   // GBK_TO_UNICODE[37068] := 16#E9F9;
   // GBK_TO_UNICODE[37069] := 16#8F7E;
   // GBK_TO_UNICODE[37070] := 16#E9FA;
   // GBK_TO_UNICODE[37071] := 16#8F81;
   // GBK_TO_UNICODE[37072] := 16#E9FB;
   // GBK_TO_UNICODE[37073] := 16#8F82;
   // GBK_TO_UNICODE[37074] := 16#E9FC;
   // GBK_TO_UNICODE[37075] := 16#8F84;
   // GBK_TO_UNICODE[37076] := 16#E9FD;
   // GBK_TO_UNICODE[37077] := 16#8F87;
   // GBK_TO_UNICODE[37078] := 16#E9FE;
   // GBK_TO_UNICODE[37079] := 16#8F8B;
   // GBK_TO_UNICODE[37080] := 16#EA40;
   // GBK_TO_UNICODE[37081] := 16#95CC;
   // GBK_TO_UNICODE[37082] := 16#EA41;
   // GBK_TO_UNICODE[37083] := 16#95CD;
   // GBK_TO_UNICODE[37084] := 16#EA42;
   // GBK_TO_UNICODE[37085] := 16#95CE;
   // GBK_TO_UNICODE[37086] := 16#EA43;
   // GBK_TO_UNICODE[37087] := 16#95CF;
   // GBK_TO_UNICODE[37088] := 16#EA44;
   // GBK_TO_UNICODE[37089] := 16#95D0;
   // GBK_TO_UNICODE[37090] := 16#EA45;
   // GBK_TO_UNICODE[37091] := 16#95D1;
   // GBK_TO_UNICODE[37092] := 16#EA46;
   // GBK_TO_UNICODE[37093] := 16#95D2;
   // GBK_TO_UNICODE[37094] := 16#EA47;
   // GBK_TO_UNICODE[37095] := 16#95D3;
   // GBK_TO_UNICODE[37096] := 16#EA48;
   // GBK_TO_UNICODE[37097] := 16#95D4;
   // GBK_TO_UNICODE[37098] := 16#EA49;
   // GBK_TO_UNICODE[37099] := 16#95D5;
   // GBK_TO_UNICODE[37100] := 16#EA4A;
   // GBK_TO_UNICODE[37101] := 16#95D6;
   // GBK_TO_UNICODE[37102] := 16#EA4B;
   // GBK_TO_UNICODE[37103] := 16#95D7;
   // GBK_TO_UNICODE[37104] := 16#EA4C;
   // GBK_TO_UNICODE[37105] := 16#95D8;
   // GBK_TO_UNICODE[37106] := 16#EA4D;
   // GBK_TO_UNICODE[37107] := 16#95D9;
   // GBK_TO_UNICODE[37108] := 16#EA4E;
   // GBK_TO_UNICODE[37109] := 16#95DA;
   // GBK_TO_UNICODE[37110] := 16#EA4F;
   // GBK_TO_UNICODE[37111] := 16#95DB;
   // GBK_TO_UNICODE[37112] := 16#EA50;
   // GBK_TO_UNICODE[37113] := 16#95DC;
   // GBK_TO_UNICODE[37114] := 16#EA51;
   // GBK_TO_UNICODE[37115] := 16#95DD;
   // GBK_TO_UNICODE[37116] := 16#EA52;
   // GBK_TO_UNICODE[37117] := 16#95DE;
   // GBK_TO_UNICODE[37118] := 16#EA53;
   // GBK_TO_UNICODE[37119] := 16#95DF;
   // GBK_TO_UNICODE[37120] := 16#EA54;
   // GBK_TO_UNICODE[37121] := 16#95E0;
   // GBK_TO_UNICODE[37122] := 16#EA55;
   // GBK_TO_UNICODE[37123] := 16#95E1;
   // GBK_TO_UNICODE[37124] := 16#EA56;
   // GBK_TO_UNICODE[37125] := 16#95E2;
   // GBK_TO_UNICODE[37126] := 16#EA57;
   // GBK_TO_UNICODE[37127] := 16#95E3;
   // GBK_TO_UNICODE[37128] := 16#EA58;
   // GBK_TO_UNICODE[37129] := 16#95E4;
   // GBK_TO_UNICODE[37130] := 16#EA59;
   // GBK_TO_UNICODE[37131] := 16#95E5;
   // GBK_TO_UNICODE[37132] := 16#EA5A;
   // GBK_TO_UNICODE[37133] := 16#95E6;
   // GBK_TO_UNICODE[37134] := 16#EA5B;
   // GBK_TO_UNICODE[37135] := 16#95E7;
   // GBK_TO_UNICODE[37136] := 16#EA5C;
   // GBK_TO_UNICODE[37137] := 16#95EC;
   // GBK_TO_UNICODE[37138] := 16#EA5D;
   // GBK_TO_UNICODE[37139] := 16#95FF;
   // GBK_TO_UNICODE[37140] := 16#EA5E;
   // GBK_TO_UNICODE[37141] := 16#9607;
   // GBK_TO_UNICODE[37142] := 16#EA5F;
   // GBK_TO_UNICODE[37143] := 16#9613;
   // GBK_TO_UNICODE[37144] := 16#EA60;
   // GBK_TO_UNICODE[37145] := 16#9618;
   // GBK_TO_UNICODE[37146] := 16#EA61;
   // GBK_TO_UNICODE[37147] := 16#961B;
   // GBK_TO_UNICODE[37148] := 16#EA62;
   // GBK_TO_UNICODE[37149] := 16#961E;
   // GBK_TO_UNICODE[37150] := 16#EA63;
   // GBK_TO_UNICODE[37151] := 16#9620;
   // GBK_TO_UNICODE[37152] := 16#EA64;
   // GBK_TO_UNICODE[37153] := 16#9623;
   // GBK_TO_UNICODE[37154] := 16#EA65;
   // GBK_TO_UNICODE[37155] := 16#9624;
   // GBK_TO_UNICODE[37156] := 16#EA66;
   // GBK_TO_UNICODE[37157] := 16#9625;
   // GBK_TO_UNICODE[37158] := 16#EA67;
   // GBK_TO_UNICODE[37159] := 16#9626;
   // GBK_TO_UNICODE[37160] := 16#EA68;
   // GBK_TO_UNICODE[37161] := 16#9627;
   // GBK_TO_UNICODE[37162] := 16#EA69;
   // GBK_TO_UNICODE[37163] := 16#9628;
   // GBK_TO_UNICODE[37164] := 16#EA6A;
   // GBK_TO_UNICODE[37165] := 16#9629;
   // GBK_TO_UNICODE[37166] := 16#EA6B;
   // GBK_TO_UNICODE[37167] := 16#962B;
   // GBK_TO_UNICODE[37168] := 16#EA6C;
   // GBK_TO_UNICODE[37169] := 16#962C;
   // GBK_TO_UNICODE[37170] := 16#EA6D;
   // GBK_TO_UNICODE[37171] := 16#962D;
   // GBK_TO_UNICODE[37172] := 16#EA6E;
   // GBK_TO_UNICODE[37173] := 16#962F;
   // GBK_TO_UNICODE[37174] := 16#EA6F;
   // GBK_TO_UNICODE[37175] := 16#9630;
   // GBK_TO_UNICODE[37176] := 16#EA70;
   // GBK_TO_UNICODE[37177] := 16#9637;
   // GBK_TO_UNICODE[37178] := 16#EA71;
   // GBK_TO_UNICODE[37179] := 16#9638;
   // GBK_TO_UNICODE[37180] := 16#EA72;
   // GBK_TO_UNICODE[37181] := 16#9639;
   // GBK_TO_UNICODE[37182] := 16#EA73;
   // GBK_TO_UNICODE[37183] := 16#963A;
   // GBK_TO_UNICODE[37184] := 16#EA74;
   // GBK_TO_UNICODE[37185] := 16#963E;
   // GBK_TO_UNICODE[37186] := 16#EA75;
   // GBK_TO_UNICODE[37187] := 16#9641;
   // GBK_TO_UNICODE[37188] := 16#EA76;
   // GBK_TO_UNICODE[37189] := 16#9643;
   // GBK_TO_UNICODE[37190] := 16#EA77;
   // GBK_TO_UNICODE[37191] := 16#964A;
   // GBK_TO_UNICODE[37192] := 16#EA78;
   // GBK_TO_UNICODE[37193] := 16#964E;
   // GBK_TO_UNICODE[37194] := 16#EA79;
   // GBK_TO_UNICODE[37195] := 16#964F;
   // GBK_TO_UNICODE[37196] := 16#EA7A;
   // GBK_TO_UNICODE[37197] := 16#9651;
   // GBK_TO_UNICODE[37198] := 16#EA7B;
   // GBK_TO_UNICODE[37199] := 16#9652;
   // GBK_TO_UNICODE[37200] := 16#EA7C;
   // GBK_TO_UNICODE[37201] := 16#9653;
   // GBK_TO_UNICODE[37202] := 16#EA7D;
   // GBK_TO_UNICODE[37203] := 16#9656;
   // GBK_TO_UNICODE[37204] := 16#EA7E;
   // GBK_TO_UNICODE[37205] := 16#9657;
   // GBK_TO_UNICODE[37206] := 16#EA80;
   // GBK_TO_UNICODE[37207] := 16#9658;
   // GBK_TO_UNICODE[37208] := 16#EA81;
   // GBK_TO_UNICODE[37209] := 16#9659;
   // GBK_TO_UNICODE[37210] := 16#EA82;
   // GBK_TO_UNICODE[37211] := 16#965A;
   // GBK_TO_UNICODE[37212] := 16#EA83;
   // GBK_TO_UNICODE[37213] := 16#965C;
   // GBK_TO_UNICODE[37214] := 16#EA84;
   // GBK_TO_UNICODE[37215] := 16#965D;
   // GBK_TO_UNICODE[37216] := 16#EA85;
   // GBK_TO_UNICODE[37217] := 16#965E;
   // GBK_TO_UNICODE[37218] := 16#EA86;
   // GBK_TO_UNICODE[37219] := 16#9660;
   // GBK_TO_UNICODE[37220] := 16#EA87;
   // GBK_TO_UNICODE[37221] := 16#9663;
   // GBK_TO_UNICODE[37222] := 16#EA88;
   // GBK_TO_UNICODE[37223] := 16#9665;
   // GBK_TO_UNICODE[37224] := 16#EA89;
   // GBK_TO_UNICODE[37225] := 16#9666;
   // GBK_TO_UNICODE[37226] := 16#EA8A;
   // GBK_TO_UNICODE[37227] := 16#966B;
   // GBK_TO_UNICODE[37228] := 16#EA8B;
   // GBK_TO_UNICODE[37229] := 16#966D;
   // GBK_TO_UNICODE[37230] := 16#EA8C;
   // GBK_TO_UNICODE[37231] := 16#966E;
   // GBK_TO_UNICODE[37232] := 16#EA8D;
   // GBK_TO_UNICODE[37233] := 16#966F;
   // GBK_TO_UNICODE[37234] := 16#EA8E;
   // GBK_TO_UNICODE[37235] := 16#9670;
   // GBK_TO_UNICODE[37236] := 16#EA8F;
   // GBK_TO_UNICODE[37237] := 16#9671;
   // GBK_TO_UNICODE[37238] := 16#EA90;
   // GBK_TO_UNICODE[37239] := 16#9673;
   // GBK_TO_UNICODE[37240] := 16#EA91;
   // GBK_TO_UNICODE[37241] := 16#9678;
   // GBK_TO_UNICODE[37242] := 16#EA92;
   // GBK_TO_UNICODE[37243] := 16#9679;
   // GBK_TO_UNICODE[37244] := 16#EA93;
   // GBK_TO_UNICODE[37245] := 16#967A;
   // GBK_TO_UNICODE[37246] := 16#EA94;
   // GBK_TO_UNICODE[37247] := 16#967B;
   // GBK_TO_UNICODE[37248] := 16#EA95;
   // GBK_TO_UNICODE[37249] := 16#967C;
   // GBK_TO_UNICODE[37250] := 16#EA96;
   // GBK_TO_UNICODE[37251] := 16#967D;
   // GBK_TO_UNICODE[37252] := 16#EA97;
   // GBK_TO_UNICODE[37253] := 16#967E;
   // GBK_TO_UNICODE[37254] := 16#EA98;
   // GBK_TO_UNICODE[37255] := 16#967F;
   // GBK_TO_UNICODE[37256] := 16#EA99;
   // GBK_TO_UNICODE[37257] := 16#9680;
   // GBK_TO_UNICODE[37258] := 16#EA9A;
   // GBK_TO_UNICODE[37259] := 16#9681;
   // GBK_TO_UNICODE[37260] := 16#EA9B;
   // GBK_TO_UNICODE[37261] := 16#9682;
   // GBK_TO_UNICODE[37262] := 16#EA9C;
   // GBK_TO_UNICODE[37263] := 16#9683;
   // GBK_TO_UNICODE[37264] := 16#EA9D;
   // GBK_TO_UNICODE[37265] := 16#9684;
   // GBK_TO_UNICODE[37266] := 16#EA9E;
   // GBK_TO_UNICODE[37267] := 16#9687;
   // GBK_TO_UNICODE[37268] := 16#EA9F;
   // GBK_TO_UNICODE[37269] := 16#9689;
   // GBK_TO_UNICODE[37270] := 16#EAA0;
   // GBK_TO_UNICODE[37271] := 16#968A;
   // GBK_TO_UNICODE[37272] := 16#EAA1;
   // GBK_TO_UNICODE[37273] := 16#8F8D;
   // GBK_TO_UNICODE[37274] := 16#EAA2;
   // GBK_TO_UNICODE[37275] := 16#8F8E;
   // GBK_TO_UNICODE[37276] := 16#EAA3;
   // GBK_TO_UNICODE[37277] := 16#8F8F;
   // GBK_TO_UNICODE[37278] := 16#EAA4;
   // GBK_TO_UNICODE[37279] := 16#8F98;
   // GBK_TO_UNICODE[37280] := 16#EAA5;
   // GBK_TO_UNICODE[37281] := 16#8F9A;
   // GBK_TO_UNICODE[37282] := 16#EAA6;
   // GBK_TO_UNICODE[37283] := 16#8ECE;
   // GBK_TO_UNICODE[37284] := 16#EAA7;
   // GBK_TO_UNICODE[37285] := 16#620B;
   // GBK_TO_UNICODE[37286] := 16#EAA8;
   // GBK_TO_UNICODE[37287] := 16#6217;
   // GBK_TO_UNICODE[37288] := 16#EAA9;
   // GBK_TO_UNICODE[37289] := 16#621B;
   // GBK_TO_UNICODE[37290] := 16#EAAA;
   // GBK_TO_UNICODE[37291] := 16#621F;
   // GBK_TO_UNICODE[37292] := 16#EAAB;
   // GBK_TO_UNICODE[37293] := 16#6222;
   // GBK_TO_UNICODE[37294] := 16#EAAC;
   // GBK_TO_UNICODE[37295] := 16#6221;
   // GBK_TO_UNICODE[37296] := 16#EAAD;
   // GBK_TO_UNICODE[37297] := 16#6225;
   // GBK_TO_UNICODE[37298] := 16#EAAE;
   // GBK_TO_UNICODE[37299] := 16#6224;
   // GBK_TO_UNICODE[37300] := 16#EAAF;
   // GBK_TO_UNICODE[37301] := 16#622C;
   // GBK_TO_UNICODE[37302] := 16#EAB0;
   // GBK_TO_UNICODE[37303] := 16#81E7;
   // GBK_TO_UNICODE[37304] := 16#EAB1;
   // GBK_TO_UNICODE[37305] := 16#74EF;
   // GBK_TO_UNICODE[37306] := 16#EAB2;
   // GBK_TO_UNICODE[37307] := 16#74F4;
   // GBK_TO_UNICODE[37308] := 16#EAB3;
   // GBK_TO_UNICODE[37309] := 16#74FF;
   // GBK_TO_UNICODE[37310] := 16#EAB4;
   // GBK_TO_UNICODE[37311] := 16#750F;
   // GBK_TO_UNICODE[37312] := 16#EAB5;
   // GBK_TO_UNICODE[37313] := 16#7511;
   // GBK_TO_UNICODE[37314] := 16#EAB6;
   // GBK_TO_UNICODE[37315] := 16#7513;
   // GBK_TO_UNICODE[37316] := 16#EAB7;
   // GBK_TO_UNICODE[37317] := 16#6534;
   // GBK_TO_UNICODE[37318] := 16#EAB8;
   // GBK_TO_UNICODE[37319] := 16#65EE;
   // GBK_TO_UNICODE[37320] := 16#EAB9;
   // GBK_TO_UNICODE[37321] := 16#65EF;
   // GBK_TO_UNICODE[37322] := 16#EABA;
   // GBK_TO_UNICODE[37323] := 16#65F0;
   // GBK_TO_UNICODE[37324] := 16#EABB;
   // GBK_TO_UNICODE[37325] := 16#660A;
   // GBK_TO_UNICODE[37326] := 16#EABC;
   // GBK_TO_UNICODE[37327] := 16#6619;
   // GBK_TO_UNICODE[37328] := 16#EABD;
   // GBK_TO_UNICODE[37329] := 16#6772;
   // GBK_TO_UNICODE[37330] := 16#EABE;
   // GBK_TO_UNICODE[37331] := 16#6603;
   // GBK_TO_UNICODE[37332] := 16#EABF;
   // GBK_TO_UNICODE[37333] := 16#6615;
   // GBK_TO_UNICODE[37334] := 16#EAC0;
   // GBK_TO_UNICODE[37335] := 16#6600;
   // GBK_TO_UNICODE[37336] := 16#EAC1;
   // GBK_TO_UNICODE[37337] := 16#7085;
   // GBK_TO_UNICODE[37338] := 16#EAC2;
   // GBK_TO_UNICODE[37339] := 16#66F7;
   // GBK_TO_UNICODE[37340] := 16#EAC3;
   // GBK_TO_UNICODE[37341] := 16#661D;
   // GBK_TO_UNICODE[37342] := 16#EAC4;
   // GBK_TO_UNICODE[37343] := 16#6634;
   // GBK_TO_UNICODE[37344] := 16#EAC5;
   // GBK_TO_UNICODE[37345] := 16#6631;
   // GBK_TO_UNICODE[37346] := 16#EAC6;
   // GBK_TO_UNICODE[37347] := 16#6636;
   // GBK_TO_UNICODE[37348] := 16#EAC7;
   // GBK_TO_UNICODE[37349] := 16#6635;
   // GBK_TO_UNICODE[37350] := 16#EAC8;
   // GBK_TO_UNICODE[37351] := 16#8006;
   // GBK_TO_UNICODE[37352] := 16#EAC9;
   // GBK_TO_UNICODE[37353] := 16#665F;
   // GBK_TO_UNICODE[37354] := 16#EACA;
   // GBK_TO_UNICODE[37355] := 16#6654;
   // GBK_TO_UNICODE[37356] := 16#EACB;
   // GBK_TO_UNICODE[37357] := 16#6641;
   // GBK_TO_UNICODE[37358] := 16#EACC;
   // GBK_TO_UNICODE[37359] := 16#664F;
   // GBK_TO_UNICODE[37360] := 16#EACD;
   // GBK_TO_UNICODE[37361] := 16#6656;
   // GBK_TO_UNICODE[37362] := 16#EACE;
   // GBK_TO_UNICODE[37363] := 16#6661;
   // GBK_TO_UNICODE[37364] := 16#EACF;
   // GBK_TO_UNICODE[37365] := 16#6657;
   // GBK_TO_UNICODE[37366] := 16#EAD0;
   // GBK_TO_UNICODE[37367] := 16#6677;
   // GBK_TO_UNICODE[37368] := 16#EAD1;
   // GBK_TO_UNICODE[37369] := 16#6684;
   // GBK_TO_UNICODE[37370] := 16#EAD2;
   // GBK_TO_UNICODE[37371] := 16#668C;
   // GBK_TO_UNICODE[37372] := 16#EAD3;
   // GBK_TO_UNICODE[37373] := 16#66A7;
   // GBK_TO_UNICODE[37374] := 16#EAD4;
   // GBK_TO_UNICODE[37375] := 16#669D;
   // GBK_TO_UNICODE[37376] := 16#EAD5;
   // GBK_TO_UNICODE[37377] := 16#66BE;
   // GBK_TO_UNICODE[37378] := 16#EAD6;
   // GBK_TO_UNICODE[37379] := 16#66DB;
   // GBK_TO_UNICODE[37380] := 16#EAD7;
   // GBK_TO_UNICODE[37381] := 16#66DC;
   // GBK_TO_UNICODE[37382] := 16#EAD8;
   // GBK_TO_UNICODE[37383] := 16#66E6;
   // GBK_TO_UNICODE[37384] := 16#EAD9;
   // GBK_TO_UNICODE[37385] := 16#66E9;
   // GBK_TO_UNICODE[37386] := 16#EADA;
   // GBK_TO_UNICODE[37387] := 16#8D32;
   // GBK_TO_UNICODE[37388] := 16#EADB;
   // GBK_TO_UNICODE[37389] := 16#8D33;
   // GBK_TO_UNICODE[37390] := 16#EADC;
   // GBK_TO_UNICODE[37391] := 16#8D36;
   // GBK_TO_UNICODE[37392] := 16#EADD;
   // GBK_TO_UNICODE[37393] := 16#8D3B;
   // GBK_TO_UNICODE[37394] := 16#EADE;
   // GBK_TO_UNICODE[37395] := 16#8D3D;
   // GBK_TO_UNICODE[37396] := 16#EADF;
   // GBK_TO_UNICODE[37397] := 16#8D40;
   // GBK_TO_UNICODE[37398] := 16#EAE0;
   // GBK_TO_UNICODE[37399] := 16#8D45;
   // GBK_TO_UNICODE[37400] := 16#EAE1;
   // GBK_TO_UNICODE[37401] := 16#8D46;
   // GBK_TO_UNICODE[37402] := 16#EAE2;
   // GBK_TO_UNICODE[37403] := 16#8D48;
   // GBK_TO_UNICODE[37404] := 16#EAE3;
   // GBK_TO_UNICODE[37405] := 16#8D49;
   // GBK_TO_UNICODE[37406] := 16#EAE4;
   // GBK_TO_UNICODE[37407] := 16#8D47;
   // GBK_TO_UNICODE[37408] := 16#EAE5;
   // GBK_TO_UNICODE[37409] := 16#8D4D;
   // GBK_TO_UNICODE[37410] := 16#EAE6;
   // GBK_TO_UNICODE[37411] := 16#8D55;
   // GBK_TO_UNICODE[37412] := 16#EAE7;
   // GBK_TO_UNICODE[37413] := 16#8D59;
   // GBK_TO_UNICODE[37414] := 16#EAE8;
   // GBK_TO_UNICODE[37415] := 16#89C7;
   // GBK_TO_UNICODE[37416] := 16#EAE9;
   // GBK_TO_UNICODE[37417] := 16#89CA;
   // GBK_TO_UNICODE[37418] := 16#EAEA;
   // GBK_TO_UNICODE[37419] := 16#89CB;
   // GBK_TO_UNICODE[37420] := 16#EAEB;
   // GBK_TO_UNICODE[37421] := 16#89CC;
   // GBK_TO_UNICODE[37422] := 16#EAEC;
   // GBK_TO_UNICODE[37423] := 16#89CE;
   // GBK_TO_UNICODE[37424] := 16#EAED;
   // GBK_TO_UNICODE[37425] := 16#89CF;
   // GBK_TO_UNICODE[37426] := 16#EAEE;
   // GBK_TO_UNICODE[37427] := 16#89D0;
   // GBK_TO_UNICODE[37428] := 16#EAEF;
   // GBK_TO_UNICODE[37429] := 16#89D1;
   // GBK_TO_UNICODE[37430] := 16#EAF0;
   // GBK_TO_UNICODE[37431] := 16#726E;
   // GBK_TO_UNICODE[37432] := 16#EAF1;
   // GBK_TO_UNICODE[37433] := 16#729F;
   // GBK_TO_UNICODE[37434] := 16#EAF2;
   // GBK_TO_UNICODE[37435] := 16#725D;
   // GBK_TO_UNICODE[37436] := 16#EAF3;
   // GBK_TO_UNICODE[37437] := 16#7266;
   // GBK_TO_UNICODE[37438] := 16#EAF4;
   // GBK_TO_UNICODE[37439] := 16#726F;
   // GBK_TO_UNICODE[37440] := 16#EAF5;
   // GBK_TO_UNICODE[37441] := 16#727E;
   // GBK_TO_UNICODE[37442] := 16#EAF6;
   // GBK_TO_UNICODE[37443] := 16#727F;
   // GBK_TO_UNICODE[37444] := 16#EAF7;
   // GBK_TO_UNICODE[37445] := 16#7284;
   // GBK_TO_UNICODE[37446] := 16#EAF8;
   // GBK_TO_UNICODE[37447] := 16#728B;
   // GBK_TO_UNICODE[37448] := 16#EAF9;
   // GBK_TO_UNICODE[37449] := 16#728D;
   // GBK_TO_UNICODE[37450] := 16#EAFA;
   // GBK_TO_UNICODE[37451] := 16#728F;
   // GBK_TO_UNICODE[37452] := 16#EAFB;
   // GBK_TO_UNICODE[37453] := 16#7292;
   // GBK_TO_UNICODE[37454] := 16#EAFC;
   // GBK_TO_UNICODE[37455] := 16#6308;
   // GBK_TO_UNICODE[37456] := 16#EAFD;
   // GBK_TO_UNICODE[37457] := 16#6332;
   // GBK_TO_UNICODE[37458] := 16#EAFE;
   // GBK_TO_UNICODE[37459] := 16#63B0;
   // GBK_TO_UNICODE[37460] := 16#EB40;
   // GBK_TO_UNICODE[37461] := 16#968C;
   // GBK_TO_UNICODE[37462] := 16#EB41;
   // GBK_TO_UNICODE[37463] := 16#968E;
   // GBK_TO_UNICODE[37464] := 16#EB42;
   // GBK_TO_UNICODE[37465] := 16#9691;
   // GBK_TO_UNICODE[37466] := 16#EB43;
   // GBK_TO_UNICODE[37467] := 16#9692;
   // GBK_TO_UNICODE[37468] := 16#EB44;
   // GBK_TO_UNICODE[37469] := 16#9693;
   // GBK_TO_UNICODE[37470] := 16#EB45;
   // GBK_TO_UNICODE[37471] := 16#9695;
   // GBK_TO_UNICODE[37472] := 16#EB46;
   // GBK_TO_UNICODE[37473] := 16#9696;
   // GBK_TO_UNICODE[37474] := 16#EB47;
   // GBK_TO_UNICODE[37475] := 16#969A;
   // GBK_TO_UNICODE[37476] := 16#EB48;
   // GBK_TO_UNICODE[37477] := 16#969B;
   // GBK_TO_UNICODE[37478] := 16#EB49;
   // GBK_TO_UNICODE[37479] := 16#969D;
   // GBK_TO_UNICODE[37480] := 16#EB4A;
   // GBK_TO_UNICODE[37481] := 16#969E;
   // GBK_TO_UNICODE[37482] := 16#EB4B;
   // GBK_TO_UNICODE[37483] := 16#969F;
   // GBK_TO_UNICODE[37484] := 16#EB4C;
   // GBK_TO_UNICODE[37485] := 16#96A0;
   // GBK_TO_UNICODE[37486] := 16#EB4D;
   // GBK_TO_UNICODE[37487] := 16#96A1;
   // GBK_TO_UNICODE[37488] := 16#EB4E;
   // GBK_TO_UNICODE[37489] := 16#96A2;
   // GBK_TO_UNICODE[37490] := 16#EB4F;
   // GBK_TO_UNICODE[37491] := 16#96A3;
   // GBK_TO_UNICODE[37492] := 16#EB50;
   // GBK_TO_UNICODE[37493] := 16#96A4;
   // GBK_TO_UNICODE[37494] := 16#EB51;
   // GBK_TO_UNICODE[37495] := 16#96A5;
   // GBK_TO_UNICODE[37496] := 16#EB52;
   // GBK_TO_UNICODE[37497] := 16#96A6;
   // GBK_TO_UNICODE[37498] := 16#EB53;
   // GBK_TO_UNICODE[37499] := 16#96A8;
   // GBK_TO_UNICODE[37500] := 16#EB54;
   // GBK_TO_UNICODE[37501] := 16#96A9;
   // GBK_TO_UNICODE[37502] := 16#EB55;
   // GBK_TO_UNICODE[37503] := 16#96AA;
   // GBK_TO_UNICODE[37504] := 16#EB56;
   // GBK_TO_UNICODE[37505] := 16#96AB;
   // GBK_TO_UNICODE[37506] := 16#EB57;
   // GBK_TO_UNICODE[37507] := 16#96AC;
   // GBK_TO_UNICODE[37508] := 16#EB58;
   // GBK_TO_UNICODE[37509] := 16#96AD;
   // GBK_TO_UNICODE[37510] := 16#EB59;
   // GBK_TO_UNICODE[37511] := 16#96AE;
   // GBK_TO_UNICODE[37512] := 16#EB5A;
   // GBK_TO_UNICODE[37513] := 16#96AF;
   // GBK_TO_UNICODE[37514] := 16#EB5B;
   // GBK_TO_UNICODE[37515] := 16#96B1;
   // GBK_TO_UNICODE[37516] := 16#EB5C;
   // GBK_TO_UNICODE[37517] := 16#96B2;
   // GBK_TO_UNICODE[37518] := 16#EB5D;
   // GBK_TO_UNICODE[37519] := 16#96B4;
   // GBK_TO_UNICODE[37520] := 16#EB5E;
   // GBK_TO_UNICODE[37521] := 16#96B5;
   // GBK_TO_UNICODE[37522] := 16#EB5F;
   // GBK_TO_UNICODE[37523] := 16#96B7;
   // GBK_TO_UNICODE[37524] := 16#EB60;
   // GBK_TO_UNICODE[37525] := 16#96B8;
   // GBK_TO_UNICODE[37526] := 16#EB61;
   // GBK_TO_UNICODE[37527] := 16#96BA;
   // GBK_TO_UNICODE[37528] := 16#EB62;
   // GBK_TO_UNICODE[37529] := 16#96BB;
   // GBK_TO_UNICODE[37530] := 16#EB63;
   // GBK_TO_UNICODE[37531] := 16#96BF;
   // GBK_TO_UNICODE[37532] := 16#EB64;
   // GBK_TO_UNICODE[37533] := 16#96C2;
   // GBK_TO_UNICODE[37534] := 16#EB65;
   // GBK_TO_UNICODE[37535] := 16#96C3;
   // GBK_TO_UNICODE[37536] := 16#EB66;
   // GBK_TO_UNICODE[37537] := 16#96C8;
   // GBK_TO_UNICODE[37538] := 16#EB67;
   // GBK_TO_UNICODE[37539] := 16#96CA;
   // GBK_TO_UNICODE[37540] := 16#EB68;
   // GBK_TO_UNICODE[37541] := 16#96CB;
   // GBK_TO_UNICODE[37542] := 16#EB69;
   // GBK_TO_UNICODE[37543] := 16#96D0;
   // GBK_TO_UNICODE[37544] := 16#EB6A;
   // GBK_TO_UNICODE[37545] := 16#96D1;
   // GBK_TO_UNICODE[37546] := 16#EB6B;
   // GBK_TO_UNICODE[37547] := 16#96D3;
   // GBK_TO_UNICODE[37548] := 16#EB6C;
   // GBK_TO_UNICODE[37549] := 16#96D4;
   // GBK_TO_UNICODE[37550] := 16#EB6D;
   // GBK_TO_UNICODE[37551] := 16#96D6;
   // GBK_TO_UNICODE[37552] := 16#EB6E;
   // GBK_TO_UNICODE[37553] := 16#96D7;
   // GBK_TO_UNICODE[37554] := 16#EB6F;
   // GBK_TO_UNICODE[37555] := 16#96D8;
   // GBK_TO_UNICODE[37556] := 16#EB70;
   // GBK_TO_UNICODE[37557] := 16#96D9;
   // GBK_TO_UNICODE[37558] := 16#EB71;
   // GBK_TO_UNICODE[37559] := 16#96DA;
   // GBK_TO_UNICODE[37560] := 16#EB72;
   // GBK_TO_UNICODE[37561] := 16#96DB;
   // GBK_TO_UNICODE[37562] := 16#EB73;
   // GBK_TO_UNICODE[37563] := 16#96DC;
   // GBK_TO_UNICODE[37564] := 16#EB74;
   // GBK_TO_UNICODE[37565] := 16#96DD;
   // GBK_TO_UNICODE[37566] := 16#EB75;
   // GBK_TO_UNICODE[37567] := 16#96DE;
   // GBK_TO_UNICODE[37568] := 16#EB76;
   // GBK_TO_UNICODE[37569] := 16#96DF;
   // GBK_TO_UNICODE[37570] := 16#EB77;
   // GBK_TO_UNICODE[37571] := 16#96E1;
   // GBK_TO_UNICODE[37572] := 16#EB78;
   // GBK_TO_UNICODE[37573] := 16#96E2;
   // GBK_TO_UNICODE[37574] := 16#EB79;
   // GBK_TO_UNICODE[37575] := 16#96E3;
   // GBK_TO_UNICODE[37576] := 16#EB7A;
   // GBK_TO_UNICODE[37577] := 16#96E4;
   // GBK_TO_UNICODE[37578] := 16#EB7B;
   // GBK_TO_UNICODE[37579] := 16#96E5;
   // GBK_TO_UNICODE[37580] := 16#EB7C;
   // GBK_TO_UNICODE[37581] := 16#96E6;
   // GBK_TO_UNICODE[37582] := 16#EB7D;
   // GBK_TO_UNICODE[37583] := 16#96E7;
   // GBK_TO_UNICODE[37584] := 16#EB7E;
   // GBK_TO_UNICODE[37585] := 16#96EB;
   // GBK_TO_UNICODE[37586] := 16#EB80;
   // GBK_TO_UNICODE[37587] := 16#96EC;
   // GBK_TO_UNICODE[37588] := 16#EB81;
   // GBK_TO_UNICODE[37589] := 16#96ED;
   // GBK_TO_UNICODE[37590] := 16#EB82;
   // GBK_TO_UNICODE[37591] := 16#96EE;
   // GBK_TO_UNICODE[37592] := 16#EB83;
   // GBK_TO_UNICODE[37593] := 16#96F0;
   // GBK_TO_UNICODE[37594] := 16#EB84;
   // GBK_TO_UNICODE[37595] := 16#96F1;
   // GBK_TO_UNICODE[37596] := 16#EB85;
   // GBK_TO_UNICODE[37597] := 16#96F2;
   // GBK_TO_UNICODE[37598] := 16#EB86;
   // GBK_TO_UNICODE[37599] := 16#96F4;
   // GBK_TO_UNICODE[37600] := 16#EB87;
   // GBK_TO_UNICODE[37601] := 16#96F5;
   // GBK_TO_UNICODE[37602] := 16#EB88;
   // GBK_TO_UNICODE[37603] := 16#96F8;
   // GBK_TO_UNICODE[37604] := 16#EB89;
   // GBK_TO_UNICODE[37605] := 16#96FA;
   // GBK_TO_UNICODE[37606] := 16#EB8A;
   // GBK_TO_UNICODE[37607] := 16#96FB;
   // GBK_TO_UNICODE[37608] := 16#EB8B;
   // GBK_TO_UNICODE[37609] := 16#96FC;
   // GBK_TO_UNICODE[37610] := 16#EB8C;
   // GBK_TO_UNICODE[37611] := 16#96FD;
   // GBK_TO_UNICODE[37612] := 16#EB8D;
   // GBK_TO_UNICODE[37613] := 16#96FF;
   // GBK_TO_UNICODE[37614] := 16#EB8E;
   // GBK_TO_UNICODE[37615] := 16#9702;
   // GBK_TO_UNICODE[37616] := 16#EB8F;
   // GBK_TO_UNICODE[37617] := 16#9703;
   // GBK_TO_UNICODE[37618] := 16#EB90;
   // GBK_TO_UNICODE[37619] := 16#9705;
   // GBK_TO_UNICODE[37620] := 16#EB91;
   // GBK_TO_UNICODE[37621] := 16#970A;
   // GBK_TO_UNICODE[37622] := 16#EB92;
   // GBK_TO_UNICODE[37623] := 16#970B;
   // GBK_TO_UNICODE[37624] := 16#EB93;
   // GBK_TO_UNICODE[37625] := 16#970C;
   // GBK_TO_UNICODE[37626] := 16#EB94;
   // GBK_TO_UNICODE[37627] := 16#9710;
   // GBK_TO_UNICODE[37628] := 16#EB95;
   // GBK_TO_UNICODE[37629] := 16#9711;
   // GBK_TO_UNICODE[37630] := 16#EB96;
   // GBK_TO_UNICODE[37631] := 16#9712;
   // GBK_TO_UNICODE[37632] := 16#EB97;
   // GBK_TO_UNICODE[37633] := 16#9714;
   // GBK_TO_UNICODE[37634] := 16#EB98;
   // GBK_TO_UNICODE[37635] := 16#9715;
   // GBK_TO_UNICODE[37636] := 16#EB99;
   // GBK_TO_UNICODE[37637] := 16#9717;
   // GBK_TO_UNICODE[37638] := 16#EB9A;
   // GBK_TO_UNICODE[37639] := 16#9718;
   // GBK_TO_UNICODE[37640] := 16#EB9B;
   // GBK_TO_UNICODE[37641] := 16#9719;
   // GBK_TO_UNICODE[37642] := 16#EB9C;
   // GBK_TO_UNICODE[37643] := 16#971A;
   // GBK_TO_UNICODE[37644] := 16#EB9D;
   // GBK_TO_UNICODE[37645] := 16#971B;
   // GBK_TO_UNICODE[37646] := 16#EB9E;
   // GBK_TO_UNICODE[37647] := 16#971D;
   // GBK_TO_UNICODE[37648] := 16#EB9F;
   // GBK_TO_UNICODE[37649] := 16#971F;
   // GBK_TO_UNICODE[37650] := 16#EBA0;
   // GBK_TO_UNICODE[37651] := 16#9720;
   // GBK_TO_UNICODE[37652] := 16#EBA1;
   // GBK_TO_UNICODE[37653] := 16#643F;
   // GBK_TO_UNICODE[37654] := 16#EBA2;
   // GBK_TO_UNICODE[37655] := 16#64D8;
   // GBK_TO_UNICODE[37656] := 16#EBA3;
   // GBK_TO_UNICODE[37657] := 16#8004;
   // GBK_TO_UNICODE[37658] := 16#EBA4;
   // GBK_TO_UNICODE[37659] := 16#6BEA;
   // GBK_TO_UNICODE[37660] := 16#EBA5;
   // GBK_TO_UNICODE[37661] := 16#6BF3;
   // GBK_TO_UNICODE[37662] := 16#EBA6;
   // GBK_TO_UNICODE[37663] := 16#6BFD;
   // GBK_TO_UNICODE[37664] := 16#EBA7;
   // GBK_TO_UNICODE[37665] := 16#6BF5;
   // GBK_TO_UNICODE[37666] := 16#EBA8;
   // GBK_TO_UNICODE[37667] := 16#6BF9;
   // GBK_TO_UNICODE[37668] := 16#EBA9;
   // GBK_TO_UNICODE[37669] := 16#6C05;
   // GBK_TO_UNICODE[37670] := 16#EBAA;
   // GBK_TO_UNICODE[37671] := 16#6C07;
   // GBK_TO_UNICODE[37672] := 16#EBAB;
   // GBK_TO_UNICODE[37673] := 16#6C06;
   // GBK_TO_UNICODE[37674] := 16#EBAC;
   // GBK_TO_UNICODE[37675] := 16#6C0D;
   // GBK_TO_UNICODE[37676] := 16#EBAD;
   // GBK_TO_UNICODE[37677] := 16#6C15;
   // GBK_TO_UNICODE[37678] := 16#EBAE;
   // GBK_TO_UNICODE[37679] := 16#6C18;
   // GBK_TO_UNICODE[37680] := 16#EBAF;
   // GBK_TO_UNICODE[37681] := 16#6C19;
   // GBK_TO_UNICODE[37682] := 16#EBB0;
   // GBK_TO_UNICODE[37683] := 16#6C1A;
   // GBK_TO_UNICODE[37684] := 16#EBB1;
   // GBK_TO_UNICODE[37685] := 16#6C21;
   // GBK_TO_UNICODE[37686] := 16#EBB2;
   // GBK_TO_UNICODE[37687] := 16#6C29;
   // GBK_TO_UNICODE[37688] := 16#EBB3;
   // GBK_TO_UNICODE[37689] := 16#6C24;
   // GBK_TO_UNICODE[37690] := 16#EBB4;
   // GBK_TO_UNICODE[37691] := 16#6C2A;
   // GBK_TO_UNICODE[37692] := 16#EBB5;
   // GBK_TO_UNICODE[37693] := 16#6C32;
   // GBK_TO_UNICODE[37694] := 16#EBB6;
   // GBK_TO_UNICODE[37695] := 16#6535;
   // GBK_TO_UNICODE[37696] := 16#EBB7;
   // GBK_TO_UNICODE[37697] := 16#6555;
   // GBK_TO_UNICODE[37698] := 16#EBB8;
   // GBK_TO_UNICODE[37699] := 16#656B;
   // GBK_TO_UNICODE[37700] := 16#EBB9;
   // GBK_TO_UNICODE[37701] := 16#724D;
   // GBK_TO_UNICODE[37702] := 16#EBBA;
   // GBK_TO_UNICODE[37703] := 16#7252;
   // GBK_TO_UNICODE[37704] := 16#EBBB;
   // GBK_TO_UNICODE[37705] := 16#7256;
   // GBK_TO_UNICODE[37706] := 16#EBBC;
   // GBK_TO_UNICODE[37707] := 16#7230;
   // GBK_TO_UNICODE[37708] := 16#EBBD;
   // GBK_TO_UNICODE[37709] := 16#8662;
   // GBK_TO_UNICODE[37710] := 16#EBBE;
   // GBK_TO_UNICODE[37711] := 16#5216;
   // GBK_TO_UNICODE[37712] := 16#EBBF;
   // GBK_TO_UNICODE[37713] := 16#809F;
   // GBK_TO_UNICODE[37714] := 16#EBC0;
   // GBK_TO_UNICODE[37715] := 16#809C;
   // GBK_TO_UNICODE[37716] := 16#EBC1;
   // GBK_TO_UNICODE[37717] := 16#8093;
   // GBK_TO_UNICODE[37718] := 16#EBC2;
   // GBK_TO_UNICODE[37719] := 16#80BC;
   // GBK_TO_UNICODE[37720] := 16#EBC3;
   // GBK_TO_UNICODE[37721] := 16#670A;
   // GBK_TO_UNICODE[37722] := 16#EBC4;
   // GBK_TO_UNICODE[37723] := 16#80BD;
   // GBK_TO_UNICODE[37724] := 16#EBC5;
   // GBK_TO_UNICODE[37725] := 16#80B1;
   // GBK_TO_UNICODE[37726] := 16#EBC6;
   // GBK_TO_UNICODE[37727] := 16#80AB;
   // GBK_TO_UNICODE[37728] := 16#EBC7;
   // GBK_TO_UNICODE[37729] := 16#80AD;
   // GBK_TO_UNICODE[37730] := 16#EBC8;
   // GBK_TO_UNICODE[37731] := 16#80B4;
   // GBK_TO_UNICODE[37732] := 16#EBC9;
   // GBK_TO_UNICODE[37733] := 16#80B7;
   // GBK_TO_UNICODE[37734] := 16#EBCA;
   // GBK_TO_UNICODE[37735] := 16#80E7;
   // GBK_TO_UNICODE[37736] := 16#EBCB;
   // GBK_TO_UNICODE[37737] := 16#80E8;
   // GBK_TO_UNICODE[37738] := 16#EBCC;
   // GBK_TO_UNICODE[37739] := 16#80E9;
   // GBK_TO_UNICODE[37740] := 16#EBCD;
   // GBK_TO_UNICODE[37741] := 16#80EA;
   // GBK_TO_UNICODE[37742] := 16#EBCE;
   // GBK_TO_UNICODE[37743] := 16#80DB;
   // GBK_TO_UNICODE[37744] := 16#EBCF;
   // GBK_TO_UNICODE[37745] := 16#80C2;
   // GBK_TO_UNICODE[37746] := 16#EBD0;
   // GBK_TO_UNICODE[37747] := 16#80C4;
   // GBK_TO_UNICODE[37748] := 16#EBD1;
   // GBK_TO_UNICODE[37749] := 16#80D9;
   // GBK_TO_UNICODE[37750] := 16#EBD2;
   // GBK_TO_UNICODE[37751] := 16#80CD;
   // GBK_TO_UNICODE[37752] := 16#EBD3;
   // GBK_TO_UNICODE[37753] := 16#80D7;
   // GBK_TO_UNICODE[37754] := 16#EBD4;
   // GBK_TO_UNICODE[37755] := 16#6710;
   // GBK_TO_UNICODE[37756] := 16#EBD5;
   // GBK_TO_UNICODE[37757] := 16#80DD;
   // GBK_TO_UNICODE[37758] := 16#EBD6;
   // GBK_TO_UNICODE[37759] := 16#80EB;
   // GBK_TO_UNICODE[37760] := 16#EBD7;
   // GBK_TO_UNICODE[37761] := 16#80F1;
   // GBK_TO_UNICODE[37762] := 16#EBD8;
   // GBK_TO_UNICODE[37763] := 16#80F4;
   // GBK_TO_UNICODE[37764] := 16#EBD9;
   // GBK_TO_UNICODE[37765] := 16#80ED;
   // GBK_TO_UNICODE[37766] := 16#EBDA;
   // GBK_TO_UNICODE[37767] := 16#810D;
   // GBK_TO_UNICODE[37768] := 16#EBDB;
   // GBK_TO_UNICODE[37769] := 16#810E;
   // GBK_TO_UNICODE[37770] := 16#EBDC;
   // GBK_TO_UNICODE[37771] := 16#80F2;
   // GBK_TO_UNICODE[37772] := 16#EBDD;
   // GBK_TO_UNICODE[37773] := 16#80FC;
   // GBK_TO_UNICODE[37774] := 16#EBDE;
   // GBK_TO_UNICODE[37775] := 16#6715;
   // GBK_TO_UNICODE[37776] := 16#EBDF;
   // GBK_TO_UNICODE[37777] := 16#8112;
   // GBK_TO_UNICODE[37778] := 16#EBE0;
   // GBK_TO_UNICODE[37779] := 16#8C5A;
   // GBK_TO_UNICODE[37780] := 16#EBE1;
   // GBK_TO_UNICODE[37781] := 16#8136;
   // GBK_TO_UNICODE[37782] := 16#EBE2;
   // GBK_TO_UNICODE[37783] := 16#811E;
   // GBK_TO_UNICODE[37784] := 16#EBE3;
   // GBK_TO_UNICODE[37785] := 16#812C;
   // GBK_TO_UNICODE[37786] := 16#EBE4;
   // GBK_TO_UNICODE[37787] := 16#8118;
   // GBK_TO_UNICODE[37788] := 16#EBE5;
   // GBK_TO_UNICODE[37789] := 16#8132;
   // GBK_TO_UNICODE[37790] := 16#EBE6;
   // GBK_TO_UNICODE[37791] := 16#8148;
   // GBK_TO_UNICODE[37792] := 16#EBE7;
   // GBK_TO_UNICODE[37793] := 16#814C;
   // GBK_TO_UNICODE[37794] := 16#EBE8;
   // GBK_TO_UNICODE[37795] := 16#8153;
   // GBK_TO_UNICODE[37796] := 16#EBE9;
   // GBK_TO_UNICODE[37797] := 16#8174;
   // GBK_TO_UNICODE[37798] := 16#EBEA;
   // GBK_TO_UNICODE[37799] := 16#8159;
   // GBK_TO_UNICODE[37800] := 16#EBEB;
   // GBK_TO_UNICODE[37801] := 16#815A;
   // GBK_TO_UNICODE[37802] := 16#EBEC;
   // GBK_TO_UNICODE[37803] := 16#8171;
   // GBK_TO_UNICODE[37804] := 16#EBED;
   // GBK_TO_UNICODE[37805] := 16#8160;
   // GBK_TO_UNICODE[37806] := 16#EBEE;
   // GBK_TO_UNICODE[37807] := 16#8169;
   // GBK_TO_UNICODE[37808] := 16#EBEF;
   // GBK_TO_UNICODE[37809] := 16#817C;
   // GBK_TO_UNICODE[37810] := 16#EBF0;
   // GBK_TO_UNICODE[37811] := 16#817D;
   // GBK_TO_UNICODE[37812] := 16#EBF1;
   // GBK_TO_UNICODE[37813] := 16#816D;
   // GBK_TO_UNICODE[37814] := 16#EBF2;
   // GBK_TO_UNICODE[37815] := 16#8167;
   // GBK_TO_UNICODE[37816] := 16#EBF3;
   // GBK_TO_UNICODE[37817] := 16#584D;
   // GBK_TO_UNICODE[37818] := 16#EBF4;
   // GBK_TO_UNICODE[37819] := 16#5AB5;
   // GBK_TO_UNICODE[37820] := 16#EBF5;
   // GBK_TO_UNICODE[37821] := 16#8188;
   // GBK_TO_UNICODE[37822] := 16#EBF6;
   // GBK_TO_UNICODE[37823] := 16#8182;
   // GBK_TO_UNICODE[37824] := 16#EBF7;
   // GBK_TO_UNICODE[37825] := 16#8191;
   // GBK_TO_UNICODE[37826] := 16#EBF8;
   // GBK_TO_UNICODE[37827] := 16#6ED5;
   // GBK_TO_UNICODE[37828] := 16#EBF9;
   // GBK_TO_UNICODE[37829] := 16#81A3;
   // GBK_TO_UNICODE[37830] := 16#EBFA;
   // GBK_TO_UNICODE[37831] := 16#81AA;
   // GBK_TO_UNICODE[37832] := 16#EBFB;
   // GBK_TO_UNICODE[37833] := 16#81CC;
   // GBK_TO_UNICODE[37834] := 16#EBFC;
   // GBK_TO_UNICODE[37835] := 16#6726;
   // GBK_TO_UNICODE[37836] := 16#EBFD;
   // GBK_TO_UNICODE[37837] := 16#81CA;
   // GBK_TO_UNICODE[37838] := 16#EBFE;
   // GBK_TO_UNICODE[37839] := 16#81BB;
   // GBK_TO_UNICODE[37840] := 16#EC40;
   // GBK_TO_UNICODE[37841] := 16#9721;
   // GBK_TO_UNICODE[37842] := 16#EC41;
   // GBK_TO_UNICODE[37843] := 16#9722;
   // GBK_TO_UNICODE[37844] := 16#EC42;
   // GBK_TO_UNICODE[37845] := 16#9723;
   // GBK_TO_UNICODE[37846] := 16#EC43;
   // GBK_TO_UNICODE[37847] := 16#9724;
   // GBK_TO_UNICODE[37848] := 16#EC44;
   // GBK_TO_UNICODE[37849] := 16#9725;
   // GBK_TO_UNICODE[37850] := 16#EC45;
   // GBK_TO_UNICODE[37851] := 16#9726;
   // GBK_TO_UNICODE[37852] := 16#EC46;
   // GBK_TO_UNICODE[37853] := 16#9727;
   // GBK_TO_UNICODE[37854] := 16#EC47;
   // GBK_TO_UNICODE[37855] := 16#9728;
   // GBK_TO_UNICODE[37856] := 16#EC48;
   // GBK_TO_UNICODE[37857] := 16#9729;
   // GBK_TO_UNICODE[37858] := 16#EC49;
   // GBK_TO_UNICODE[37859] := 16#972B;
   // GBK_TO_UNICODE[37860] := 16#EC4A;
   // GBK_TO_UNICODE[37861] := 16#972C;
   // GBK_TO_UNICODE[37862] := 16#EC4B;
   // GBK_TO_UNICODE[37863] := 16#972E;
   // GBK_TO_UNICODE[37864] := 16#EC4C;
   // GBK_TO_UNICODE[37865] := 16#972F;
   // GBK_TO_UNICODE[37866] := 16#EC4D;
   // GBK_TO_UNICODE[37867] := 16#9731;
   // GBK_TO_UNICODE[37868] := 16#EC4E;
   // GBK_TO_UNICODE[37869] := 16#9733;
   // GBK_TO_UNICODE[37870] := 16#EC4F;
   // GBK_TO_UNICODE[37871] := 16#9734;
   // GBK_TO_UNICODE[37872] := 16#EC50;
   // GBK_TO_UNICODE[37873] := 16#9735;
   // GBK_TO_UNICODE[37874] := 16#EC51;
   // GBK_TO_UNICODE[37875] := 16#9736;
   // GBK_TO_UNICODE[37876] := 16#EC52;
   // GBK_TO_UNICODE[37877] := 16#9737;
   // GBK_TO_UNICODE[37878] := 16#EC53;
   // GBK_TO_UNICODE[37879] := 16#973A;
   // GBK_TO_UNICODE[37880] := 16#EC54;
   // GBK_TO_UNICODE[37881] := 16#973B;
   // GBK_TO_UNICODE[37882] := 16#EC55;
   // GBK_TO_UNICODE[37883] := 16#973C;
   // GBK_TO_UNICODE[37884] := 16#EC56;
   // GBK_TO_UNICODE[37885] := 16#973D;
   // GBK_TO_UNICODE[37886] := 16#EC57;
   // GBK_TO_UNICODE[37887] := 16#973F;
   // GBK_TO_UNICODE[37888] := 16#EC58;
   // GBK_TO_UNICODE[37889] := 16#9740;
   // GBK_TO_UNICODE[37890] := 16#EC59;
   // GBK_TO_UNICODE[37891] := 16#9741;
   // GBK_TO_UNICODE[37892] := 16#EC5A;
   // GBK_TO_UNICODE[37893] := 16#9742;
   // GBK_TO_UNICODE[37894] := 16#EC5B;
   // GBK_TO_UNICODE[37895] := 16#9743;
   // GBK_TO_UNICODE[37896] := 16#EC5C;
   // GBK_TO_UNICODE[37897] := 16#9744;
   // GBK_TO_UNICODE[37898] := 16#EC5D;
   // GBK_TO_UNICODE[37899] := 16#9745;
   // GBK_TO_UNICODE[37900] := 16#EC5E;
   // GBK_TO_UNICODE[37901] := 16#9746;
   // GBK_TO_UNICODE[37902] := 16#EC5F;
   // GBK_TO_UNICODE[37903] := 16#9747;
   // GBK_TO_UNICODE[37904] := 16#EC60;
   // GBK_TO_UNICODE[37905] := 16#9748;
   // GBK_TO_UNICODE[37906] := 16#EC61;
   // GBK_TO_UNICODE[37907] := 16#9749;
   // GBK_TO_UNICODE[37908] := 16#EC62;
   // GBK_TO_UNICODE[37909] := 16#974A;
   // GBK_TO_UNICODE[37910] := 16#EC63;
   // GBK_TO_UNICODE[37911] := 16#974B;
   // GBK_TO_UNICODE[37912] := 16#EC64;
   // GBK_TO_UNICODE[37913] := 16#974C;
   // GBK_TO_UNICODE[37914] := 16#EC65;
   // GBK_TO_UNICODE[37915] := 16#974D;
   // GBK_TO_UNICODE[37916] := 16#EC66;
   // GBK_TO_UNICODE[37917] := 16#974E;
   // GBK_TO_UNICODE[37918] := 16#EC67;
   // GBK_TO_UNICODE[37919] := 16#974F;
   // GBK_TO_UNICODE[37920] := 16#EC68;
   // GBK_TO_UNICODE[37921] := 16#9750;
   // GBK_TO_UNICODE[37922] := 16#EC69;
   // GBK_TO_UNICODE[37923] := 16#9751;
   // GBK_TO_UNICODE[37924] := 16#EC6A;
   // GBK_TO_UNICODE[37925] := 16#9754;
   // GBK_TO_UNICODE[37926] := 16#EC6B;
   // GBK_TO_UNICODE[37927] := 16#9755;
   // GBK_TO_UNICODE[37928] := 16#EC6C;
   // GBK_TO_UNICODE[37929] := 16#9757;
   // GBK_TO_UNICODE[37930] := 16#EC6D;
   // GBK_TO_UNICODE[37931] := 16#9758;
   // GBK_TO_UNICODE[37932] := 16#EC6E;
   // GBK_TO_UNICODE[37933] := 16#975A;
   // GBK_TO_UNICODE[37934] := 16#EC6F;
   // GBK_TO_UNICODE[37935] := 16#975C;
   // GBK_TO_UNICODE[37936] := 16#EC70;
   // GBK_TO_UNICODE[37937] := 16#975D;
   // GBK_TO_UNICODE[37938] := 16#EC71;
   // GBK_TO_UNICODE[37939] := 16#975F;
   // GBK_TO_UNICODE[37940] := 16#EC72;
   // GBK_TO_UNICODE[37941] := 16#9763;
   // GBK_TO_UNICODE[37942] := 16#EC73;
   // GBK_TO_UNICODE[37943] := 16#9764;
   // GBK_TO_UNICODE[37944] := 16#EC74;
   // GBK_TO_UNICODE[37945] := 16#9766;
   // GBK_TO_UNICODE[37946] := 16#EC75;
   // GBK_TO_UNICODE[37947] := 16#9767;
   // GBK_TO_UNICODE[37948] := 16#EC76;
   // GBK_TO_UNICODE[37949] := 16#9768;
   // GBK_TO_UNICODE[37950] := 16#EC77;
   // GBK_TO_UNICODE[37951] := 16#976A;
   // GBK_TO_UNICODE[37952] := 16#EC78;
   // GBK_TO_UNICODE[37953] := 16#976B;
   // GBK_TO_UNICODE[37954] := 16#EC79;
   // GBK_TO_UNICODE[37955] := 16#976C;
   // GBK_TO_UNICODE[37956] := 16#EC7A;
   // GBK_TO_UNICODE[37957] := 16#976D;
   // GBK_TO_UNICODE[37958] := 16#EC7B;
   // GBK_TO_UNICODE[37959] := 16#976E;
   // GBK_TO_UNICODE[37960] := 16#EC7C;
   // GBK_TO_UNICODE[37961] := 16#976F;
   // GBK_TO_UNICODE[37962] := 16#EC7D;
   // GBK_TO_UNICODE[37963] := 16#9770;
   // GBK_TO_UNICODE[37964] := 16#EC7E;
   // GBK_TO_UNICODE[37965] := 16#9771;
   // GBK_TO_UNICODE[37966] := 16#EC80;
   // GBK_TO_UNICODE[37967] := 16#9772;
   // GBK_TO_UNICODE[37968] := 16#EC81;
   // GBK_TO_UNICODE[37969] := 16#9775;
   // GBK_TO_UNICODE[37970] := 16#EC82;
   // GBK_TO_UNICODE[37971] := 16#9777;
   // GBK_TO_UNICODE[37972] := 16#EC83;
   // GBK_TO_UNICODE[37973] := 16#9778;
   // GBK_TO_UNICODE[37974] := 16#EC84;
   // GBK_TO_UNICODE[37975] := 16#9779;
   // GBK_TO_UNICODE[37976] := 16#EC85;
   // GBK_TO_UNICODE[37977] := 16#977A;
   // GBK_TO_UNICODE[37978] := 16#EC86;
   // GBK_TO_UNICODE[37979] := 16#977B;
   // GBK_TO_UNICODE[37980] := 16#EC87;
   // GBK_TO_UNICODE[37981] := 16#977D;
   // GBK_TO_UNICODE[37982] := 16#EC88;
   // GBK_TO_UNICODE[37983] := 16#977E;
   // GBK_TO_UNICODE[37984] := 16#EC89;
   // GBK_TO_UNICODE[37985] := 16#977F;
   // GBK_TO_UNICODE[37986] := 16#EC8A;
   // GBK_TO_UNICODE[37987] := 16#9780;
   // GBK_TO_UNICODE[37988] := 16#EC8B;
   // GBK_TO_UNICODE[37989] := 16#9781;
   // GBK_TO_UNICODE[37990] := 16#EC8C;
   // GBK_TO_UNICODE[37991] := 16#9782;
   // GBK_TO_UNICODE[37992] := 16#EC8D;
   // GBK_TO_UNICODE[37993] := 16#9783;
   // GBK_TO_UNICODE[37994] := 16#EC8E;
   // GBK_TO_UNICODE[37995] := 16#9784;
   // GBK_TO_UNICODE[37996] := 16#EC8F;
   // GBK_TO_UNICODE[37997] := 16#9786;
   // GBK_TO_UNICODE[37998] := 16#EC90;
   // GBK_TO_UNICODE[37999] := 16#9787;
   // GBK_TO_UNICODE[38000] := 16#EC91;
   // GBK_TO_UNICODE[38001] := 16#9788;
   // GBK_TO_UNICODE[38002] := 16#EC92;
   // GBK_TO_UNICODE[38003] := 16#9789;
   // GBK_TO_UNICODE[38004] := 16#EC93;
   // GBK_TO_UNICODE[38005] := 16#978A;
   // GBK_TO_UNICODE[38006] := 16#EC94;
   // GBK_TO_UNICODE[38007] := 16#978C;
   // GBK_TO_UNICODE[38008] := 16#EC95;
   // GBK_TO_UNICODE[38009] := 16#978E;
   // GBK_TO_UNICODE[38010] := 16#EC96;
   // GBK_TO_UNICODE[38011] := 16#978F;
   // GBK_TO_UNICODE[38012] := 16#EC97;
   // GBK_TO_UNICODE[38013] := 16#9790;
   // GBK_TO_UNICODE[38014] := 16#EC98;
   // GBK_TO_UNICODE[38015] := 16#9793;
   // GBK_TO_UNICODE[38016] := 16#EC99;
   // GBK_TO_UNICODE[38017] := 16#9795;
   // GBK_TO_UNICODE[38018] := 16#EC9A;
   // GBK_TO_UNICODE[38019] := 16#9796;
   // GBK_TO_UNICODE[38020] := 16#EC9B;
   // GBK_TO_UNICODE[38021] := 16#9797;
   // GBK_TO_UNICODE[38022] := 16#EC9C;
   // GBK_TO_UNICODE[38023] := 16#9799;
   // GBK_TO_UNICODE[38024] := 16#EC9D;
   // GBK_TO_UNICODE[38025] := 16#979A;
   // GBK_TO_UNICODE[38026] := 16#EC9E;
   // GBK_TO_UNICODE[38027] := 16#979B;
   // GBK_TO_UNICODE[38028] := 16#EC9F;
   // GBK_TO_UNICODE[38029] := 16#979C;
   // GBK_TO_UNICODE[38030] := 16#ECA0;
   // GBK_TO_UNICODE[38031] := 16#979D;
   // GBK_TO_UNICODE[38032] := 16#ECA1;
   // GBK_TO_UNICODE[38033] := 16#81C1;
   // GBK_TO_UNICODE[38034] := 16#ECA2;
   // GBK_TO_UNICODE[38035] := 16#81A6;
   // GBK_TO_UNICODE[38036] := 16#ECA3;
   // GBK_TO_UNICODE[38037] := 16#6B24;
   // GBK_TO_UNICODE[38038] := 16#ECA4;
   // GBK_TO_UNICODE[38039] := 16#6B37;
   // GBK_TO_UNICODE[38040] := 16#ECA5;
   // GBK_TO_UNICODE[38041] := 16#6B39;
   // GBK_TO_UNICODE[38042] := 16#ECA6;
   // GBK_TO_UNICODE[38043] := 16#6B43;
   // GBK_TO_UNICODE[38044] := 16#ECA7;
   // GBK_TO_UNICODE[38045] := 16#6B46;
   // GBK_TO_UNICODE[38046] := 16#ECA8;
   // GBK_TO_UNICODE[38047] := 16#6B59;
   // GBK_TO_UNICODE[38048] := 16#ECA9;
   // GBK_TO_UNICODE[38049] := 16#98D1;
   // GBK_TO_UNICODE[38050] := 16#ECAA;
   // GBK_TO_UNICODE[38051] := 16#98D2;
   // GBK_TO_UNICODE[38052] := 16#ECAB;
   // GBK_TO_UNICODE[38053] := 16#98D3;
   // GBK_TO_UNICODE[38054] := 16#ECAC;
   // GBK_TO_UNICODE[38055] := 16#98D5;
   // GBK_TO_UNICODE[38056] := 16#ECAD;
   // GBK_TO_UNICODE[38057] := 16#98D9;
   // GBK_TO_UNICODE[38058] := 16#ECAE;
   // GBK_TO_UNICODE[38059] := 16#98DA;
   // GBK_TO_UNICODE[38060] := 16#ECAF;
   // GBK_TO_UNICODE[38061] := 16#6BB3;
   // GBK_TO_UNICODE[38062] := 16#ECB0;
   // GBK_TO_UNICODE[38063] := 16#5F40;
   // GBK_TO_UNICODE[38064] := 16#ECB1;
   // GBK_TO_UNICODE[38065] := 16#6BC2;
   // GBK_TO_UNICODE[38066] := 16#ECB2;
   // GBK_TO_UNICODE[38067] := 16#89F3;
   // GBK_TO_UNICODE[38068] := 16#ECB3;
   // GBK_TO_UNICODE[38069] := 16#6590;
   // GBK_TO_UNICODE[38070] := 16#ECB4;
   // GBK_TO_UNICODE[38071] := 16#9F51;
   // GBK_TO_UNICODE[38072] := 16#ECB5;
   // GBK_TO_UNICODE[38073] := 16#6593;
   // GBK_TO_UNICODE[38074] := 16#ECB6;
   // GBK_TO_UNICODE[38075] := 16#65BC;
   // GBK_TO_UNICODE[38076] := 16#ECB7;
   // GBK_TO_UNICODE[38077] := 16#65C6;
   // GBK_TO_UNICODE[38078] := 16#ECB8;
   // GBK_TO_UNICODE[38079] := 16#65C4;
   // GBK_TO_UNICODE[38080] := 16#ECB9;
   // GBK_TO_UNICODE[38081] := 16#65C3;
   // GBK_TO_UNICODE[38082] := 16#ECBA;
   // GBK_TO_UNICODE[38083] := 16#65CC;
   // GBK_TO_UNICODE[38084] := 16#ECBB;
   // GBK_TO_UNICODE[38085] := 16#65CE;
   // GBK_TO_UNICODE[38086] := 16#ECBC;
   // GBK_TO_UNICODE[38087] := 16#65D2;
   // GBK_TO_UNICODE[38088] := 16#ECBD;
   // GBK_TO_UNICODE[38089] := 16#65D6;
   // GBK_TO_UNICODE[38090] := 16#ECBE;
   // GBK_TO_UNICODE[38091] := 16#7080;
   // GBK_TO_UNICODE[38092] := 16#ECBF;
   // GBK_TO_UNICODE[38093] := 16#709C;
   // GBK_TO_UNICODE[38094] := 16#ECC0;
   // GBK_TO_UNICODE[38095] := 16#7096;
   // GBK_TO_UNICODE[38096] := 16#ECC1;
   // GBK_TO_UNICODE[38097] := 16#709D;
   // GBK_TO_UNICODE[38098] := 16#ECC2;
   // GBK_TO_UNICODE[38099] := 16#70BB;
   // GBK_TO_UNICODE[38100] := 16#ECC3;
   // GBK_TO_UNICODE[38101] := 16#70C0;
   // GBK_TO_UNICODE[38102] := 16#ECC4;
   // GBK_TO_UNICODE[38103] := 16#70B7;
   // GBK_TO_UNICODE[38104] := 16#ECC5;
   // GBK_TO_UNICODE[38105] := 16#70AB;
   // GBK_TO_UNICODE[38106] := 16#ECC6;
   // GBK_TO_UNICODE[38107] := 16#70B1;
   // GBK_TO_UNICODE[38108] := 16#ECC7;
   // GBK_TO_UNICODE[38109] := 16#70E8;
   // GBK_TO_UNICODE[38110] := 16#ECC8;
   // GBK_TO_UNICODE[38111] := 16#70CA;
   // GBK_TO_UNICODE[38112] := 16#ECC9;
   // GBK_TO_UNICODE[38113] := 16#7110;
   // GBK_TO_UNICODE[38114] := 16#ECCA;
   // GBK_TO_UNICODE[38115] := 16#7113;
   // GBK_TO_UNICODE[38116] := 16#ECCB;
   // GBK_TO_UNICODE[38117] := 16#7116;
   // GBK_TO_UNICODE[38118] := 16#ECCC;
   // GBK_TO_UNICODE[38119] := 16#712F;
   // GBK_TO_UNICODE[38120] := 16#ECCD;
   // GBK_TO_UNICODE[38121] := 16#7131;
   // GBK_TO_UNICODE[38122] := 16#ECCE;
   // GBK_TO_UNICODE[38123] := 16#7173;
   // GBK_TO_UNICODE[38124] := 16#ECCF;
   // GBK_TO_UNICODE[38125] := 16#715C;
   // GBK_TO_UNICODE[38126] := 16#ECD0;
   // GBK_TO_UNICODE[38127] := 16#7168;
   // GBK_TO_UNICODE[38128] := 16#ECD1;
   // GBK_TO_UNICODE[38129] := 16#7145;
   // GBK_TO_UNICODE[38130] := 16#ECD2;
   // GBK_TO_UNICODE[38131] := 16#7172;
   // GBK_TO_UNICODE[38132] := 16#ECD3;
   // GBK_TO_UNICODE[38133] := 16#714A;
   // GBK_TO_UNICODE[38134] := 16#ECD4;
   // GBK_TO_UNICODE[38135] := 16#7178;
   // GBK_TO_UNICODE[38136] := 16#ECD5;
   // GBK_TO_UNICODE[38137] := 16#717A;
   // GBK_TO_UNICODE[38138] := 16#ECD6;
   // GBK_TO_UNICODE[38139] := 16#7198;
   // GBK_TO_UNICODE[38140] := 16#ECD7;
   // GBK_TO_UNICODE[38141] := 16#71B3;
   // GBK_TO_UNICODE[38142] := 16#ECD8;
   // GBK_TO_UNICODE[38143] := 16#71B5;
   // GBK_TO_UNICODE[38144] := 16#ECD9;
   // GBK_TO_UNICODE[38145] := 16#71A8;
   // GBK_TO_UNICODE[38146] := 16#ECDA;
   // GBK_TO_UNICODE[38147] := 16#71A0;
   // GBK_TO_UNICODE[38148] := 16#ECDB;
   // GBK_TO_UNICODE[38149] := 16#71E0;
   // GBK_TO_UNICODE[38150] := 16#ECDC;
   // GBK_TO_UNICODE[38151] := 16#71D4;
   // GBK_TO_UNICODE[38152] := 16#ECDD;
   // GBK_TO_UNICODE[38153] := 16#71E7;
   // GBK_TO_UNICODE[38154] := 16#ECDE;
   // GBK_TO_UNICODE[38155] := 16#71F9;
   // GBK_TO_UNICODE[38156] := 16#ECDF;
   // GBK_TO_UNICODE[38157] := 16#721D;
   // GBK_TO_UNICODE[38158] := 16#ECE0;
   // GBK_TO_UNICODE[38159] := 16#7228;
   // GBK_TO_UNICODE[38160] := 16#ECE1;
   // GBK_TO_UNICODE[38161] := 16#706C;
   // GBK_TO_UNICODE[38162] := 16#ECE2;
   // GBK_TO_UNICODE[38163] := 16#7118;
   // GBK_TO_UNICODE[38164] := 16#ECE3;
   // GBK_TO_UNICODE[38165] := 16#7166;
   // GBK_TO_UNICODE[38166] := 16#ECE4;
   // GBK_TO_UNICODE[38167] := 16#71B9;
   // GBK_TO_UNICODE[38168] := 16#ECE5;
   // GBK_TO_UNICODE[38169] := 16#623E;
   // GBK_TO_UNICODE[38170] := 16#ECE6;
   // GBK_TO_UNICODE[38171] := 16#623D;
   // GBK_TO_UNICODE[38172] := 16#ECE7;
   // GBK_TO_UNICODE[38173] := 16#6243;
   // GBK_TO_UNICODE[38174] := 16#ECE8;
   // GBK_TO_UNICODE[38175] := 16#6248;
   // GBK_TO_UNICODE[38176] := 16#ECE9;
   // GBK_TO_UNICODE[38177] := 16#6249;
   // GBK_TO_UNICODE[38178] := 16#ECEA;
   // GBK_TO_UNICODE[38179] := 16#793B;
   // GBK_TO_UNICODE[38180] := 16#ECEB;
   // GBK_TO_UNICODE[38181] := 16#7940;
   // GBK_TO_UNICODE[38182] := 16#ECEC;
   // GBK_TO_UNICODE[38183] := 16#7946;
   // GBK_TO_UNICODE[38184] := 16#ECED;
   // GBK_TO_UNICODE[38185] := 16#7949;
   // GBK_TO_UNICODE[38186] := 16#ECEE;
   // GBK_TO_UNICODE[38187] := 16#795B;
   // GBK_TO_UNICODE[38188] := 16#ECEF;
   // GBK_TO_UNICODE[38189] := 16#795C;
   // GBK_TO_UNICODE[38190] := 16#ECF0;
   // GBK_TO_UNICODE[38191] := 16#7953;
   // GBK_TO_UNICODE[38192] := 16#ECF1;
   // GBK_TO_UNICODE[38193] := 16#795A;
   // GBK_TO_UNICODE[38194] := 16#ECF2;
   // GBK_TO_UNICODE[38195] := 16#7962;
   // GBK_TO_UNICODE[38196] := 16#ECF3;
   // GBK_TO_UNICODE[38197] := 16#7957;
   // GBK_TO_UNICODE[38198] := 16#ECF4;
   // GBK_TO_UNICODE[38199] := 16#7960;
   // GBK_TO_UNICODE[38200] := 16#ECF5;
   // GBK_TO_UNICODE[38201] := 16#796F;
   // GBK_TO_UNICODE[38202] := 16#ECF6;
   // GBK_TO_UNICODE[38203] := 16#7967;
   // GBK_TO_UNICODE[38204] := 16#ECF7;
   // GBK_TO_UNICODE[38205] := 16#797A;
   // GBK_TO_UNICODE[38206] := 16#ECF8;
   // GBK_TO_UNICODE[38207] := 16#7985;
   // GBK_TO_UNICODE[38208] := 16#ECF9;
   // GBK_TO_UNICODE[38209] := 16#798A;
   // GBK_TO_UNICODE[38210] := 16#ECFA;
   // GBK_TO_UNICODE[38211] := 16#799A;
   // GBK_TO_UNICODE[38212] := 16#ECFB;
   // GBK_TO_UNICODE[38213] := 16#79A7;
   // GBK_TO_UNICODE[38214] := 16#ECFC;
   // GBK_TO_UNICODE[38215] := 16#79B3;
   // GBK_TO_UNICODE[38216] := 16#ECFD;
   // GBK_TO_UNICODE[38217] := 16#5FD1;
   // GBK_TO_UNICODE[38218] := 16#ECFE;
   // GBK_TO_UNICODE[38219] := 16#5FD0;
   // GBK_TO_UNICODE[38220] := 16#ED40;
   // GBK_TO_UNICODE[38221] := 16#979E;
   // GBK_TO_UNICODE[38222] := 16#ED41;
   // GBK_TO_UNICODE[38223] := 16#979F;
   // GBK_TO_UNICODE[38224] := 16#ED42;
   // GBK_TO_UNICODE[38225] := 16#97A1;
   // GBK_TO_UNICODE[38226] := 16#ED43;
   // GBK_TO_UNICODE[38227] := 16#97A2;
   // GBK_TO_UNICODE[38228] := 16#ED44;
   // GBK_TO_UNICODE[38229] := 16#97A4;
   // GBK_TO_UNICODE[38230] := 16#ED45;
   // GBK_TO_UNICODE[38231] := 16#97A5;
   // GBK_TO_UNICODE[38232] := 16#ED46;
   // GBK_TO_UNICODE[38233] := 16#97A6;
   // GBK_TO_UNICODE[38234] := 16#ED47;
   // GBK_TO_UNICODE[38235] := 16#97A7;
   // GBK_TO_UNICODE[38236] := 16#ED48;
   // GBK_TO_UNICODE[38237] := 16#97A8;
   // GBK_TO_UNICODE[38238] := 16#ED49;
   // GBK_TO_UNICODE[38239] := 16#97A9;
   // GBK_TO_UNICODE[38240] := 16#ED4A;
   // GBK_TO_UNICODE[38241] := 16#97AA;
   // GBK_TO_UNICODE[38242] := 16#ED4B;
   // GBK_TO_UNICODE[38243] := 16#97AC;
   // GBK_TO_UNICODE[38244] := 16#ED4C;
   // GBK_TO_UNICODE[38245] := 16#97AE;
   // GBK_TO_UNICODE[38246] := 16#ED4D;
   // GBK_TO_UNICODE[38247] := 16#97B0;
   // GBK_TO_UNICODE[38248] := 16#ED4E;
   // GBK_TO_UNICODE[38249] := 16#97B1;
   // GBK_TO_UNICODE[38250] := 16#ED4F;
   // GBK_TO_UNICODE[38251] := 16#97B3;
   // GBK_TO_UNICODE[38252] := 16#ED50;
   // GBK_TO_UNICODE[38253] := 16#97B5;
   // GBK_TO_UNICODE[38254] := 16#ED51;
   // GBK_TO_UNICODE[38255] := 16#97B6;
   // GBK_TO_UNICODE[38256] := 16#ED52;
   // GBK_TO_UNICODE[38257] := 16#97B7;
   // GBK_TO_UNICODE[38258] := 16#ED53;
   // GBK_TO_UNICODE[38259] := 16#97B8;
   // GBK_TO_UNICODE[38260] := 16#ED54;
   // GBK_TO_UNICODE[38261] := 16#97B9;
   // GBK_TO_UNICODE[38262] := 16#ED55;
   // GBK_TO_UNICODE[38263] := 16#97BA;
   // GBK_TO_UNICODE[38264] := 16#ED56;
   // GBK_TO_UNICODE[38265] := 16#97BB;
   // GBK_TO_UNICODE[38266] := 16#ED57;
   // GBK_TO_UNICODE[38267] := 16#97BC;
   // GBK_TO_UNICODE[38268] := 16#ED58;
   // GBK_TO_UNICODE[38269] := 16#97BD;
   // GBK_TO_UNICODE[38270] := 16#ED59;
   // GBK_TO_UNICODE[38271] := 16#97BE;
   // GBK_TO_UNICODE[38272] := 16#ED5A;
   // GBK_TO_UNICODE[38273] := 16#97BF;
   // GBK_TO_UNICODE[38274] := 16#ED5B;
   // GBK_TO_UNICODE[38275] := 16#97C0;
   // GBK_TO_UNICODE[38276] := 16#ED5C;
   // GBK_TO_UNICODE[38277] := 16#97C1;
   // GBK_TO_UNICODE[38278] := 16#ED5D;
   // GBK_TO_UNICODE[38279] := 16#97C2;
   // GBK_TO_UNICODE[38280] := 16#ED5E;
   // GBK_TO_UNICODE[38281] := 16#97C3;
   // GBK_TO_UNICODE[38282] := 16#ED5F;
   // GBK_TO_UNICODE[38283] := 16#97C4;
   // GBK_TO_UNICODE[38284] := 16#ED60;
   // GBK_TO_UNICODE[38285] := 16#97C5;
   // GBK_TO_UNICODE[38286] := 16#ED61;
   // GBK_TO_UNICODE[38287] := 16#97C6;
   // GBK_TO_UNICODE[38288] := 16#ED62;
   // GBK_TO_UNICODE[38289] := 16#97C7;
   // GBK_TO_UNICODE[38290] := 16#ED63;
   // GBK_TO_UNICODE[38291] := 16#97C8;
   // GBK_TO_UNICODE[38292] := 16#ED64;
   // GBK_TO_UNICODE[38293] := 16#97C9;
   // GBK_TO_UNICODE[38294] := 16#ED65;
   // GBK_TO_UNICODE[38295] := 16#97CA;
   // GBK_TO_UNICODE[38296] := 16#ED66;
   // GBK_TO_UNICODE[38297] := 16#97CB;
   // GBK_TO_UNICODE[38298] := 16#ED67;
   // GBK_TO_UNICODE[38299] := 16#97CC;
   // GBK_TO_UNICODE[38300] := 16#ED68;
   // GBK_TO_UNICODE[38301] := 16#97CD;
   // GBK_TO_UNICODE[38302] := 16#ED69;
   // GBK_TO_UNICODE[38303] := 16#97CE;
   // GBK_TO_UNICODE[38304] := 16#ED6A;
   // GBK_TO_UNICODE[38305] := 16#97CF;
   // GBK_TO_UNICODE[38306] := 16#ED6B;
   // GBK_TO_UNICODE[38307] := 16#97D0;
   // GBK_TO_UNICODE[38308] := 16#ED6C;
   // GBK_TO_UNICODE[38309] := 16#97D1;
   // GBK_TO_UNICODE[38310] := 16#ED6D;
   // GBK_TO_UNICODE[38311] := 16#97D2;
   // GBK_TO_UNICODE[38312] := 16#ED6E;
   // GBK_TO_UNICODE[38313] := 16#97D3;
   // GBK_TO_UNICODE[38314] := 16#ED6F;
   // GBK_TO_UNICODE[38315] := 16#97D4;
   // GBK_TO_UNICODE[38316] := 16#ED70;
   // GBK_TO_UNICODE[38317] := 16#97D5;
   // GBK_TO_UNICODE[38318] := 16#ED71;
   // GBK_TO_UNICODE[38319] := 16#97D6;
   // GBK_TO_UNICODE[38320] := 16#ED72;
   // GBK_TO_UNICODE[38321] := 16#97D7;
   // GBK_TO_UNICODE[38322] := 16#ED73;
   // GBK_TO_UNICODE[38323] := 16#97D8;
   // GBK_TO_UNICODE[38324] := 16#ED74;
   // GBK_TO_UNICODE[38325] := 16#97D9;
   // GBK_TO_UNICODE[38326] := 16#ED75;
   // GBK_TO_UNICODE[38327] := 16#97DA;
   // GBK_TO_UNICODE[38328] := 16#ED76;
   // GBK_TO_UNICODE[38329] := 16#97DB;
   // GBK_TO_UNICODE[38330] := 16#ED77;
   // GBK_TO_UNICODE[38331] := 16#97DC;
   // GBK_TO_UNICODE[38332] := 16#ED78;
   // GBK_TO_UNICODE[38333] := 16#97DD;
   // GBK_TO_UNICODE[38334] := 16#ED79;
   // GBK_TO_UNICODE[38335] := 16#97DE;
   // GBK_TO_UNICODE[38336] := 16#ED7A;
   // GBK_TO_UNICODE[38337] := 16#97DF;
   // GBK_TO_UNICODE[38338] := 16#ED7B;
   // GBK_TO_UNICODE[38339] := 16#97E0;
   // GBK_TO_UNICODE[38340] := 16#ED7C;
   // GBK_TO_UNICODE[38341] := 16#97E1;
   // GBK_TO_UNICODE[38342] := 16#ED7D;
   // GBK_TO_UNICODE[38343] := 16#97E2;
   // GBK_TO_UNICODE[38344] := 16#ED7E;
   // GBK_TO_UNICODE[38345] := 16#97E3;
   // GBK_TO_UNICODE[38346] := 16#ED80;
   // GBK_TO_UNICODE[38347] := 16#97E4;
   // GBK_TO_UNICODE[38348] := 16#ED81;
   // GBK_TO_UNICODE[38349] := 16#97E5;
   // GBK_TO_UNICODE[38350] := 16#ED82;
   // GBK_TO_UNICODE[38351] := 16#97E8;
   // GBK_TO_UNICODE[38352] := 16#ED83;
   // GBK_TO_UNICODE[38353] := 16#97EE;
   // GBK_TO_UNICODE[38354] := 16#ED84;
   // GBK_TO_UNICODE[38355] := 16#97EF;
   // GBK_TO_UNICODE[38356] := 16#ED85;
   // GBK_TO_UNICODE[38357] := 16#97F0;
   // GBK_TO_UNICODE[38358] := 16#ED86;
   // GBK_TO_UNICODE[38359] := 16#97F1;
   // GBK_TO_UNICODE[38360] := 16#ED87;
   // GBK_TO_UNICODE[38361] := 16#97F2;
   // GBK_TO_UNICODE[38362] := 16#ED88;
   // GBK_TO_UNICODE[38363] := 16#97F4;
   // GBK_TO_UNICODE[38364] := 16#ED89;
   // GBK_TO_UNICODE[38365] := 16#97F7;
   // GBK_TO_UNICODE[38366] := 16#ED8A;
   // GBK_TO_UNICODE[38367] := 16#97F8;
   // GBK_TO_UNICODE[38368] := 16#ED8B;
   // GBK_TO_UNICODE[38369] := 16#97F9;
   // GBK_TO_UNICODE[38370] := 16#ED8C;
   // GBK_TO_UNICODE[38371] := 16#97FA;
   // GBK_TO_UNICODE[38372] := 16#ED8D;
   // GBK_TO_UNICODE[38373] := 16#97FB;
   // GBK_TO_UNICODE[38374] := 16#ED8E;
   // GBK_TO_UNICODE[38375] := 16#97FC;
   // GBK_TO_UNICODE[38376] := 16#ED8F;
   // GBK_TO_UNICODE[38377] := 16#97FD;
   // GBK_TO_UNICODE[38378] := 16#ED90;
   // GBK_TO_UNICODE[38379] := 16#97FE;
   // GBK_TO_UNICODE[38380] := 16#ED91;
   // GBK_TO_UNICODE[38381] := 16#97FF;
   // GBK_TO_UNICODE[38382] := 16#ED92;
   // GBK_TO_UNICODE[38383] := 16#9800;
   // GBK_TO_UNICODE[38384] := 16#ED93;
   // GBK_TO_UNICODE[38385] := 16#9801;
   // GBK_TO_UNICODE[38386] := 16#ED94;
   // GBK_TO_UNICODE[38387] := 16#9802;
   // GBK_TO_UNICODE[38388] := 16#ED95;
   // GBK_TO_UNICODE[38389] := 16#9803;
   // GBK_TO_UNICODE[38390] := 16#ED96;
   // GBK_TO_UNICODE[38391] := 16#9804;
   // GBK_TO_UNICODE[38392] := 16#ED97;
   // GBK_TO_UNICODE[38393] := 16#9805;
   // GBK_TO_UNICODE[38394] := 16#ED98;
   // GBK_TO_UNICODE[38395] := 16#9806;
   // GBK_TO_UNICODE[38396] := 16#ED99;
   // GBK_TO_UNICODE[38397] := 16#9807;
   // GBK_TO_UNICODE[38398] := 16#ED9A;
   // GBK_TO_UNICODE[38399] := 16#9808;
   // GBK_TO_UNICODE[38400] := 16#ED9B;
   // GBK_TO_UNICODE[38401] := 16#9809;
   // GBK_TO_UNICODE[38402] := 16#ED9C;
   // GBK_TO_UNICODE[38403] := 16#980A;
   // GBK_TO_UNICODE[38404] := 16#ED9D;
   // GBK_TO_UNICODE[38405] := 16#980B;
   // GBK_TO_UNICODE[38406] := 16#ED9E;
   // GBK_TO_UNICODE[38407] := 16#980C;
   // GBK_TO_UNICODE[38408] := 16#ED9F;
   // GBK_TO_UNICODE[38409] := 16#980D;
   // GBK_TO_UNICODE[38410] := 16#EDA0;
   // GBK_TO_UNICODE[38411] := 16#980E;
   // GBK_TO_UNICODE[38412] := 16#EDA1;
   // GBK_TO_UNICODE[38413] := 16#603C;
   // GBK_TO_UNICODE[38414] := 16#EDA2;
   // GBK_TO_UNICODE[38415] := 16#605D;
   // GBK_TO_UNICODE[38416] := 16#EDA3;
   // GBK_TO_UNICODE[38417] := 16#605A;
   // GBK_TO_UNICODE[38418] := 16#EDA4;
   // GBK_TO_UNICODE[38419] := 16#6067;
   // GBK_TO_UNICODE[38420] := 16#EDA5;
   // GBK_TO_UNICODE[38421] := 16#6041;
   // GBK_TO_UNICODE[38422] := 16#EDA6;
   // GBK_TO_UNICODE[38423] := 16#6059;
   // GBK_TO_UNICODE[38424] := 16#EDA7;
   // GBK_TO_UNICODE[38425] := 16#6063;
   // GBK_TO_UNICODE[38426] := 16#EDA8;
   // GBK_TO_UNICODE[38427] := 16#60AB;
   // GBK_TO_UNICODE[38428] := 16#EDA9;
   // GBK_TO_UNICODE[38429] := 16#6106;
   // GBK_TO_UNICODE[38430] := 16#EDAA;
   // GBK_TO_UNICODE[38431] := 16#610D;
   // GBK_TO_UNICODE[38432] := 16#EDAB;
   // GBK_TO_UNICODE[38433] := 16#615D;
   // GBK_TO_UNICODE[38434] := 16#EDAC;
   // GBK_TO_UNICODE[38435] := 16#61A9;
   // GBK_TO_UNICODE[38436] := 16#EDAD;
   // GBK_TO_UNICODE[38437] := 16#619D;
   // GBK_TO_UNICODE[38438] := 16#EDAE;
   // GBK_TO_UNICODE[38439] := 16#61CB;
   // GBK_TO_UNICODE[38440] := 16#EDAF;
   // GBK_TO_UNICODE[38441] := 16#61D1;
   // GBK_TO_UNICODE[38442] := 16#EDB0;
   // GBK_TO_UNICODE[38443] := 16#6206;
   // GBK_TO_UNICODE[38444] := 16#EDB1;
   // GBK_TO_UNICODE[38445] := 16#8080;
   // GBK_TO_UNICODE[38446] := 16#EDB2;
   // GBK_TO_UNICODE[38447] := 16#807F;
   // GBK_TO_UNICODE[38448] := 16#EDB3;
   // GBK_TO_UNICODE[38449] := 16#6C93;
   // GBK_TO_UNICODE[38450] := 16#EDB4;
   // GBK_TO_UNICODE[38451] := 16#6CF6;
   // GBK_TO_UNICODE[38452] := 16#EDB5;
   // GBK_TO_UNICODE[38453] := 16#6DFC;
   // GBK_TO_UNICODE[38454] := 16#EDB6;
   // GBK_TO_UNICODE[38455] := 16#77F6;
   // GBK_TO_UNICODE[38456] := 16#EDB7;
   // GBK_TO_UNICODE[38457] := 16#77F8;
   // GBK_TO_UNICODE[38458] := 16#EDB8;
   // GBK_TO_UNICODE[38459] := 16#7800;
   // GBK_TO_UNICODE[38460] := 16#EDB9;
   // GBK_TO_UNICODE[38461] := 16#7809;
   // GBK_TO_UNICODE[38462] := 16#EDBA;
   // GBK_TO_UNICODE[38463] := 16#7817;
   // GBK_TO_UNICODE[38464] := 16#EDBB;
   // GBK_TO_UNICODE[38465] := 16#7818;
   // GBK_TO_UNICODE[38466] := 16#EDBC;
   // GBK_TO_UNICODE[38467] := 16#7811;
   // GBK_TO_UNICODE[38468] := 16#EDBD;
   // GBK_TO_UNICODE[38469] := 16#65AB;
   // GBK_TO_UNICODE[38470] := 16#EDBE;
   // GBK_TO_UNICODE[38471] := 16#782D;
   // GBK_TO_UNICODE[38472] := 16#EDBF;
   // GBK_TO_UNICODE[38473] := 16#781C;
   // GBK_TO_UNICODE[38474] := 16#EDC0;
   // GBK_TO_UNICODE[38475] := 16#781D;
   // GBK_TO_UNICODE[38476] := 16#EDC1;
   // GBK_TO_UNICODE[38477] := 16#7839;
   // GBK_TO_UNICODE[38478] := 16#EDC2;
   // GBK_TO_UNICODE[38479] := 16#783A;
   // GBK_TO_UNICODE[38480] := 16#EDC3;
   // GBK_TO_UNICODE[38481] := 16#783B;
   // GBK_TO_UNICODE[38482] := 16#EDC4;
   // GBK_TO_UNICODE[38483] := 16#781F;
   // GBK_TO_UNICODE[38484] := 16#EDC5;
   // GBK_TO_UNICODE[38485] := 16#783C;
   // GBK_TO_UNICODE[38486] := 16#EDC6;
   // GBK_TO_UNICODE[38487] := 16#7825;
   // GBK_TO_UNICODE[38488] := 16#EDC7;
   // GBK_TO_UNICODE[38489] := 16#782C;
   // GBK_TO_UNICODE[38490] := 16#EDC8;
   // GBK_TO_UNICODE[38491] := 16#7823;
   // GBK_TO_UNICODE[38492] := 16#EDC9;
   // GBK_TO_UNICODE[38493] := 16#7829;
   // GBK_TO_UNICODE[38494] := 16#EDCA;
   // GBK_TO_UNICODE[38495] := 16#784E;
   // GBK_TO_UNICODE[38496] := 16#EDCB;
   // GBK_TO_UNICODE[38497] := 16#786D;
   // GBK_TO_UNICODE[38498] := 16#EDCC;
   // GBK_TO_UNICODE[38499] := 16#7856;
   // GBK_TO_UNICODE[38500] := 16#EDCD;
   // GBK_TO_UNICODE[38501] := 16#7857;
   // GBK_TO_UNICODE[38502] := 16#EDCE;
   // GBK_TO_UNICODE[38503] := 16#7826;
   // GBK_TO_UNICODE[38504] := 16#EDCF;
   // GBK_TO_UNICODE[38505] := 16#7850;
   // GBK_TO_UNICODE[38506] := 16#EDD0;
   // GBK_TO_UNICODE[38507] := 16#7847;
   // GBK_TO_UNICODE[38508] := 16#EDD1;
   // GBK_TO_UNICODE[38509] := 16#784C;
   // GBK_TO_UNICODE[38510] := 16#EDD2;
   // GBK_TO_UNICODE[38511] := 16#786A;
   // GBK_TO_UNICODE[38512] := 16#EDD3;
   // GBK_TO_UNICODE[38513] := 16#789B;
   // GBK_TO_UNICODE[38514] := 16#EDD4;
   // GBK_TO_UNICODE[38515] := 16#7893;
   // GBK_TO_UNICODE[38516] := 16#EDD5;
   // GBK_TO_UNICODE[38517] := 16#789A;
   // GBK_TO_UNICODE[38518] := 16#EDD6;
   // GBK_TO_UNICODE[38519] := 16#7887;
   // GBK_TO_UNICODE[38520] := 16#EDD7;
   // GBK_TO_UNICODE[38521] := 16#789C;
   // GBK_TO_UNICODE[38522] := 16#EDD8;
   // GBK_TO_UNICODE[38523] := 16#78A1;
   // GBK_TO_UNICODE[38524] := 16#EDD9;
   // GBK_TO_UNICODE[38525] := 16#78A3;
   // GBK_TO_UNICODE[38526] := 16#EDDA;
   // GBK_TO_UNICODE[38527] := 16#78B2;
   // GBK_TO_UNICODE[38528] := 16#EDDB;
   // GBK_TO_UNICODE[38529] := 16#78B9;
   // GBK_TO_UNICODE[38530] := 16#EDDC;
   // GBK_TO_UNICODE[38531] := 16#78A5;
   // GBK_TO_UNICODE[38532] := 16#EDDD;
   // GBK_TO_UNICODE[38533] := 16#78D4;
   // GBK_TO_UNICODE[38534] := 16#EDDE;
   // GBK_TO_UNICODE[38535] := 16#78D9;
   // GBK_TO_UNICODE[38536] := 16#EDDF;
   // GBK_TO_UNICODE[38537] := 16#78C9;
   // GBK_TO_UNICODE[38538] := 16#EDE0;
   // GBK_TO_UNICODE[38539] := 16#78EC;
   // GBK_TO_UNICODE[38540] := 16#EDE1;
   // GBK_TO_UNICODE[38541] := 16#78F2;
   // GBK_TO_UNICODE[38542] := 16#EDE2;
   // GBK_TO_UNICODE[38543] := 16#7905;
   // GBK_TO_UNICODE[38544] := 16#EDE3;
   // GBK_TO_UNICODE[38545] := 16#78F4;
   // GBK_TO_UNICODE[38546] := 16#EDE4;
   // GBK_TO_UNICODE[38547] := 16#7913;
   // GBK_TO_UNICODE[38548] := 16#EDE5;
   // GBK_TO_UNICODE[38549] := 16#7924;
   // GBK_TO_UNICODE[38550] := 16#EDE6;
   // GBK_TO_UNICODE[38551] := 16#791E;
   // GBK_TO_UNICODE[38552] := 16#EDE7;
   // GBK_TO_UNICODE[38553] := 16#7934;
   // GBK_TO_UNICODE[38554] := 16#EDE8;
   // GBK_TO_UNICODE[38555] := 16#9F9B;
   // GBK_TO_UNICODE[38556] := 16#EDE9;
   // GBK_TO_UNICODE[38557] := 16#9EF9;
   // GBK_TO_UNICODE[38558] := 16#EDEA;
   // GBK_TO_UNICODE[38559] := 16#9EFB;
   // GBK_TO_UNICODE[38560] := 16#EDEB;
   // GBK_TO_UNICODE[38561] := 16#9EFC;
   // GBK_TO_UNICODE[38562] := 16#EDEC;
   // GBK_TO_UNICODE[38563] := 16#76F1;
   // GBK_TO_UNICODE[38564] := 16#EDED;
   // GBK_TO_UNICODE[38565] := 16#7704;
   // GBK_TO_UNICODE[38566] := 16#EDEE;
   // GBK_TO_UNICODE[38567] := 16#770D;
   // GBK_TO_UNICODE[38568] := 16#EDEF;
   // GBK_TO_UNICODE[38569] := 16#76F9;
   // GBK_TO_UNICODE[38570] := 16#EDF0;
   // GBK_TO_UNICODE[38571] := 16#7707;
   // GBK_TO_UNICODE[38572] := 16#EDF1;
   // GBK_TO_UNICODE[38573] := 16#7708;
   // GBK_TO_UNICODE[38574] := 16#EDF2;
   // GBK_TO_UNICODE[38575] := 16#771A;
   // GBK_TO_UNICODE[38576] := 16#EDF3;
   // GBK_TO_UNICODE[38577] := 16#7722;
   // GBK_TO_UNICODE[38578] := 16#EDF4;
   // GBK_TO_UNICODE[38579] := 16#7719;
   // GBK_TO_UNICODE[38580] := 16#EDF5;
   // GBK_TO_UNICODE[38581] := 16#772D;
   // GBK_TO_UNICODE[38582] := 16#EDF6;
   // GBK_TO_UNICODE[38583] := 16#7726;
   // GBK_TO_UNICODE[38584] := 16#EDF7;
   // GBK_TO_UNICODE[38585] := 16#7735;
   // GBK_TO_UNICODE[38586] := 16#EDF8;
   // GBK_TO_UNICODE[38587] := 16#7738;
   // GBK_TO_UNICODE[38588] := 16#EDF9;
   // GBK_TO_UNICODE[38589] := 16#7750;
   // GBK_TO_UNICODE[38590] := 16#EDFA;
   // GBK_TO_UNICODE[38591] := 16#7751;
   // GBK_TO_UNICODE[38592] := 16#EDFB;
   // GBK_TO_UNICODE[38593] := 16#7747;
   // GBK_TO_UNICODE[38594] := 16#EDFC;
   // GBK_TO_UNICODE[38595] := 16#7743;
   // GBK_TO_UNICODE[38596] := 16#EDFD;
   // GBK_TO_UNICODE[38597] := 16#775A;
   // GBK_TO_UNICODE[38598] := 16#EDFE;
   // GBK_TO_UNICODE[38599] := 16#7768;
   // GBK_TO_UNICODE[38600] := 16#EE40;
   // GBK_TO_UNICODE[38601] := 16#980F;
   // GBK_TO_UNICODE[38602] := 16#EE41;
   // GBK_TO_UNICODE[38603] := 16#9810;
   // GBK_TO_UNICODE[38604] := 16#EE42;
   // GBK_TO_UNICODE[38605] := 16#9811;
   // GBK_TO_UNICODE[38606] := 16#EE43;
   // GBK_TO_UNICODE[38607] := 16#9812;
   // GBK_TO_UNICODE[38608] := 16#EE44;
   // GBK_TO_UNICODE[38609] := 16#9813;
   // GBK_TO_UNICODE[38610] := 16#EE45;
   // GBK_TO_UNICODE[38611] := 16#9814;
   // GBK_TO_UNICODE[38612] := 16#EE46;
   // GBK_TO_UNICODE[38613] := 16#9815;
   // GBK_TO_UNICODE[38614] := 16#EE47;
   // GBK_TO_UNICODE[38615] := 16#9816;
   // GBK_TO_UNICODE[38616] := 16#EE48;
   // GBK_TO_UNICODE[38617] := 16#9817;
   // GBK_TO_UNICODE[38618] := 16#EE49;
   // GBK_TO_UNICODE[38619] := 16#9818;
   // GBK_TO_UNICODE[38620] := 16#EE4A;
   // GBK_TO_UNICODE[38621] := 16#9819;
   // GBK_TO_UNICODE[38622] := 16#EE4B;
   // GBK_TO_UNICODE[38623] := 16#981A;
   // GBK_TO_UNICODE[38624] := 16#EE4C;
   // GBK_TO_UNICODE[38625] := 16#981B;
   // GBK_TO_UNICODE[38626] := 16#EE4D;
   // GBK_TO_UNICODE[38627] := 16#981C;
   // GBK_TO_UNICODE[38628] := 16#EE4E;
   // GBK_TO_UNICODE[38629] := 16#981D;
   // GBK_TO_UNICODE[38630] := 16#EE4F;
   // GBK_TO_UNICODE[38631] := 16#981E;
   // GBK_TO_UNICODE[38632] := 16#EE50;
   // GBK_TO_UNICODE[38633] := 16#981F;
   // GBK_TO_UNICODE[38634] := 16#EE51;
   // GBK_TO_UNICODE[38635] := 16#9820;
   // GBK_TO_UNICODE[38636] := 16#EE52;
   // GBK_TO_UNICODE[38637] := 16#9821;
   // GBK_TO_UNICODE[38638] := 16#EE53;
   // GBK_TO_UNICODE[38639] := 16#9822;
   // GBK_TO_UNICODE[38640] := 16#EE54;
   // GBK_TO_UNICODE[38641] := 16#9823;
   // GBK_TO_UNICODE[38642] := 16#EE55;
   // GBK_TO_UNICODE[38643] := 16#9824;
   // GBK_TO_UNICODE[38644] := 16#EE56;
   // GBK_TO_UNICODE[38645] := 16#9825;
   // GBK_TO_UNICODE[38646] := 16#EE57;
   // GBK_TO_UNICODE[38647] := 16#9826;
   // GBK_TO_UNICODE[38648] := 16#EE58;
   // GBK_TO_UNICODE[38649] := 16#9827;
   // GBK_TO_UNICODE[38650] := 16#EE59;
   // GBK_TO_UNICODE[38651] := 16#9828;
   // GBK_TO_UNICODE[38652] := 16#EE5A;
   // GBK_TO_UNICODE[38653] := 16#9829;
   // GBK_TO_UNICODE[38654] := 16#EE5B;
   // GBK_TO_UNICODE[38655] := 16#982A;
   // GBK_TO_UNICODE[38656] := 16#EE5C;
   // GBK_TO_UNICODE[38657] := 16#982B;
   // GBK_TO_UNICODE[38658] := 16#EE5D;
   // GBK_TO_UNICODE[38659] := 16#982C;
   // GBK_TO_UNICODE[38660] := 16#EE5E;
   // GBK_TO_UNICODE[38661] := 16#982D;
   // GBK_TO_UNICODE[38662] := 16#EE5F;
   // GBK_TO_UNICODE[38663] := 16#982E;
   // GBK_TO_UNICODE[38664] := 16#EE60;
   // GBK_TO_UNICODE[38665] := 16#982F;
   // GBK_TO_UNICODE[38666] := 16#EE61;
   // GBK_TO_UNICODE[38667] := 16#9830;
   // GBK_TO_UNICODE[38668] := 16#EE62;
   // GBK_TO_UNICODE[38669] := 16#9831;
   // GBK_TO_UNICODE[38670] := 16#EE63;
   // GBK_TO_UNICODE[38671] := 16#9832;
   // GBK_TO_UNICODE[38672] := 16#EE64;
   // GBK_TO_UNICODE[38673] := 16#9833;
   // GBK_TO_UNICODE[38674] := 16#EE65;
   // GBK_TO_UNICODE[38675] := 16#9834;
   // GBK_TO_UNICODE[38676] := 16#EE66;
   // GBK_TO_UNICODE[38677] := 16#9835;
   // GBK_TO_UNICODE[38678] := 16#EE67;
   // GBK_TO_UNICODE[38679] := 16#9836;
   // GBK_TO_UNICODE[38680] := 16#EE68;
   // GBK_TO_UNICODE[38681] := 16#9837;
   // GBK_TO_UNICODE[38682] := 16#EE69;
   // GBK_TO_UNICODE[38683] := 16#9838;
   // GBK_TO_UNICODE[38684] := 16#EE6A;
   // GBK_TO_UNICODE[38685] := 16#9839;
   // GBK_TO_UNICODE[38686] := 16#EE6B;
   // GBK_TO_UNICODE[38687] := 16#983A;
   // GBK_TO_UNICODE[38688] := 16#EE6C;
   // GBK_TO_UNICODE[38689] := 16#983B;
   // GBK_TO_UNICODE[38690] := 16#EE6D;
   // GBK_TO_UNICODE[38691] := 16#983C;
   // GBK_TO_UNICODE[38692] := 16#EE6E;
   // GBK_TO_UNICODE[38693] := 16#983D;
   // GBK_TO_UNICODE[38694] := 16#EE6F;
   // GBK_TO_UNICODE[38695] := 16#983E;
   // GBK_TO_UNICODE[38696] := 16#EE70;
   // GBK_TO_UNICODE[38697] := 16#983F;
   // GBK_TO_UNICODE[38698] := 16#EE71;
   // GBK_TO_UNICODE[38699] := 16#9840;
   // GBK_TO_UNICODE[38700] := 16#EE72;
   // GBK_TO_UNICODE[38701] := 16#9841;
   // GBK_TO_UNICODE[38702] := 16#EE73;
   // GBK_TO_UNICODE[38703] := 16#9842;
   // GBK_TO_UNICODE[38704] := 16#EE74;
   // GBK_TO_UNICODE[38705] := 16#9843;
   // GBK_TO_UNICODE[38706] := 16#EE75;
   // GBK_TO_UNICODE[38707] := 16#9844;
   // GBK_TO_UNICODE[38708] := 16#EE76;
   // GBK_TO_UNICODE[38709] := 16#9845;
   // GBK_TO_UNICODE[38710] := 16#EE77;
   // GBK_TO_UNICODE[38711] := 16#9846;
   // GBK_TO_UNICODE[38712] := 16#EE78;
   // GBK_TO_UNICODE[38713] := 16#9847;
   // GBK_TO_UNICODE[38714] := 16#EE79;
   // GBK_TO_UNICODE[38715] := 16#9848;
   // GBK_TO_UNICODE[38716] := 16#EE7A;
   // GBK_TO_UNICODE[38717] := 16#9849;
   // GBK_TO_UNICODE[38718] := 16#EE7B;
   // GBK_TO_UNICODE[38719] := 16#984A;
   // GBK_TO_UNICODE[38720] := 16#EE7C;
   // GBK_TO_UNICODE[38721] := 16#984B;
   // GBK_TO_UNICODE[38722] := 16#EE7D;
   // GBK_TO_UNICODE[38723] := 16#984C;
   // GBK_TO_UNICODE[38724] := 16#EE7E;
   // GBK_TO_UNICODE[38725] := 16#984D;
   // GBK_TO_UNICODE[38726] := 16#EE80;
   // GBK_TO_UNICODE[38727] := 16#984E;
   // GBK_TO_UNICODE[38728] := 16#EE81;
   // GBK_TO_UNICODE[38729] := 16#984F;
   // GBK_TO_UNICODE[38730] := 16#EE82;
   // GBK_TO_UNICODE[38731] := 16#9850;
   // GBK_TO_UNICODE[38732] := 16#EE83;
   // GBK_TO_UNICODE[38733] := 16#9851;
   // GBK_TO_UNICODE[38734] := 16#EE84;
   // GBK_TO_UNICODE[38735] := 16#9852;
   // GBK_TO_UNICODE[38736] := 16#EE85;
   // GBK_TO_UNICODE[38737] := 16#9853;
   // GBK_TO_UNICODE[38738] := 16#EE86;
   // GBK_TO_UNICODE[38739] := 16#9854;
   // GBK_TO_UNICODE[38740] := 16#EE87;
   // GBK_TO_UNICODE[38741] := 16#9855;
   // GBK_TO_UNICODE[38742] := 16#EE88;
   // GBK_TO_UNICODE[38743] := 16#9856;
   // GBK_TO_UNICODE[38744] := 16#EE89;
   // GBK_TO_UNICODE[38745] := 16#9857;
   // GBK_TO_UNICODE[38746] := 16#EE8A;
   // GBK_TO_UNICODE[38747] := 16#9858;
   // GBK_TO_UNICODE[38748] := 16#EE8B;
   // GBK_TO_UNICODE[38749] := 16#9859;
   // GBK_TO_UNICODE[38750] := 16#EE8C;
   // GBK_TO_UNICODE[38751] := 16#985A;
   // GBK_TO_UNICODE[38752] := 16#EE8D;
   // GBK_TO_UNICODE[38753] := 16#985B;
   // GBK_TO_UNICODE[38754] := 16#EE8E;
   // GBK_TO_UNICODE[38755] := 16#985C;
   // GBK_TO_UNICODE[38756] := 16#EE8F;
   // GBK_TO_UNICODE[38757] := 16#985D;
   // GBK_TO_UNICODE[38758] := 16#EE90;
   // GBK_TO_UNICODE[38759] := 16#985E;
   // GBK_TO_UNICODE[38760] := 16#EE91;
   // GBK_TO_UNICODE[38761] := 16#985F;
   // GBK_TO_UNICODE[38762] := 16#EE92;
   // GBK_TO_UNICODE[38763] := 16#9860;
   // GBK_TO_UNICODE[38764] := 16#EE93;
   // GBK_TO_UNICODE[38765] := 16#9861;
   // GBK_TO_UNICODE[38766] := 16#EE94;
   // GBK_TO_UNICODE[38767] := 16#9862;
   // GBK_TO_UNICODE[38768] := 16#EE95;
   // GBK_TO_UNICODE[38769] := 16#9863;
   // GBK_TO_UNICODE[38770] := 16#EE96;
   // GBK_TO_UNICODE[38771] := 16#9864;
   // GBK_TO_UNICODE[38772] := 16#EE97;
   // GBK_TO_UNICODE[38773] := 16#9865;
   // GBK_TO_UNICODE[38774] := 16#EE98;
   // GBK_TO_UNICODE[38775] := 16#9866;
   // GBK_TO_UNICODE[38776] := 16#EE99;
   // GBK_TO_UNICODE[38777] := 16#9867;
   // GBK_TO_UNICODE[38778] := 16#EE9A;
   // GBK_TO_UNICODE[38779] := 16#9868;
   // GBK_TO_UNICODE[38780] := 16#EE9B;
   // GBK_TO_UNICODE[38781] := 16#9869;
   // GBK_TO_UNICODE[38782] := 16#EE9C;
   // GBK_TO_UNICODE[38783] := 16#986A;
   // GBK_TO_UNICODE[38784] := 16#EE9D;
   // GBK_TO_UNICODE[38785] := 16#986B;
   // GBK_TO_UNICODE[38786] := 16#EE9E;
   // GBK_TO_UNICODE[38787] := 16#986C;
   // GBK_TO_UNICODE[38788] := 16#EE9F;
   // GBK_TO_UNICODE[38789] := 16#986D;
   // GBK_TO_UNICODE[38790] := 16#EEA0;
   // GBK_TO_UNICODE[38791] := 16#986E;
   // GBK_TO_UNICODE[38792] := 16#EEA1;
   // GBK_TO_UNICODE[38793] := 16#7762;
   // GBK_TO_UNICODE[38794] := 16#EEA2;
   // GBK_TO_UNICODE[38795] := 16#7765;
   // GBK_TO_UNICODE[38796] := 16#EEA3;
   // GBK_TO_UNICODE[38797] := 16#777F;
   // GBK_TO_UNICODE[38798] := 16#EEA4;
   // GBK_TO_UNICODE[38799] := 16#778D;
   // GBK_TO_UNICODE[38800] := 16#EEA5;
   // GBK_TO_UNICODE[38801] := 16#777D;
   // GBK_TO_UNICODE[38802] := 16#EEA6;
   // GBK_TO_UNICODE[38803] := 16#7780;
   // GBK_TO_UNICODE[38804] := 16#EEA7;
   // GBK_TO_UNICODE[38805] := 16#778C;
   // GBK_TO_UNICODE[38806] := 16#EEA8;
   // GBK_TO_UNICODE[38807] := 16#7791;
   // GBK_TO_UNICODE[38808] := 16#EEA9;
   // GBK_TO_UNICODE[38809] := 16#779F;
   // GBK_TO_UNICODE[38810] := 16#EEAA;
   // GBK_TO_UNICODE[38811] := 16#77A0;
   // GBK_TO_UNICODE[38812] := 16#EEAB;
   // GBK_TO_UNICODE[38813] := 16#77B0;
   // GBK_TO_UNICODE[38814] := 16#EEAC;
   // GBK_TO_UNICODE[38815] := 16#77B5;
   // GBK_TO_UNICODE[38816] := 16#EEAD;
   // GBK_TO_UNICODE[38817] := 16#77BD;
   // GBK_TO_UNICODE[38818] := 16#EEAE;
   // GBK_TO_UNICODE[38819] := 16#753A;
   // GBK_TO_UNICODE[38820] := 16#EEAF;
   // GBK_TO_UNICODE[38821] := 16#7540;
   // GBK_TO_UNICODE[38822] := 16#EEB0;
   // GBK_TO_UNICODE[38823] := 16#754E;
   // GBK_TO_UNICODE[38824] := 16#EEB1;
   // GBK_TO_UNICODE[38825] := 16#754B;
   // GBK_TO_UNICODE[38826] := 16#EEB2;
   // GBK_TO_UNICODE[38827] := 16#7548;
   // GBK_TO_UNICODE[38828] := 16#EEB3;
   // GBK_TO_UNICODE[38829] := 16#755B;
   // GBK_TO_UNICODE[38830] := 16#EEB4;
   // GBK_TO_UNICODE[38831] := 16#7572;
   // GBK_TO_UNICODE[38832] := 16#EEB5;
   // GBK_TO_UNICODE[38833] := 16#7579;
   // GBK_TO_UNICODE[38834] := 16#EEB6;
   // GBK_TO_UNICODE[38835] := 16#7583;
   // GBK_TO_UNICODE[38836] := 16#EEB7;
   // GBK_TO_UNICODE[38837] := 16#7F58;
   // GBK_TO_UNICODE[38838] := 16#EEB8;
   // GBK_TO_UNICODE[38839] := 16#7F61;
   // GBK_TO_UNICODE[38840] := 16#EEB9;
   // GBK_TO_UNICODE[38841] := 16#7F5F;
   // GBK_TO_UNICODE[38842] := 16#EEBA;
   // GBK_TO_UNICODE[38843] := 16#8A48;
   // GBK_TO_UNICODE[38844] := 16#EEBB;
   // GBK_TO_UNICODE[38845] := 16#7F68;
   // GBK_TO_UNICODE[38846] := 16#EEBC;
   // GBK_TO_UNICODE[38847] := 16#7F74;
   // GBK_TO_UNICODE[38848] := 16#EEBD;
   // GBK_TO_UNICODE[38849] := 16#7F71;
   // GBK_TO_UNICODE[38850] := 16#EEBE;
   // GBK_TO_UNICODE[38851] := 16#7F79;
   // GBK_TO_UNICODE[38852] := 16#EEBF;
   // GBK_TO_UNICODE[38853] := 16#7F81;
   // GBK_TO_UNICODE[38854] := 16#EEC0;
   // GBK_TO_UNICODE[38855] := 16#7F7E;
   // GBK_TO_UNICODE[38856] := 16#EEC1;
   // GBK_TO_UNICODE[38857] := 16#76CD;
   // GBK_TO_UNICODE[38858] := 16#EEC2;
   // GBK_TO_UNICODE[38859] := 16#76E5;
   // GBK_TO_UNICODE[38860] := 16#EEC3;
   // GBK_TO_UNICODE[38861] := 16#8832;
   // GBK_TO_UNICODE[38862] := 16#EEC4;
   // GBK_TO_UNICODE[38863] := 16#9485;
   // GBK_TO_UNICODE[38864] := 16#EEC5;
   // GBK_TO_UNICODE[38865] := 16#9486;
   // GBK_TO_UNICODE[38866] := 16#EEC6;
   // GBK_TO_UNICODE[38867] := 16#9487;
   // GBK_TO_UNICODE[38868] := 16#EEC7;
   // GBK_TO_UNICODE[38869] := 16#948B;
   // GBK_TO_UNICODE[38870] := 16#EEC8;
   // GBK_TO_UNICODE[38871] := 16#948A;
   // GBK_TO_UNICODE[38872] := 16#EEC9;
   // GBK_TO_UNICODE[38873] := 16#948C;
   // GBK_TO_UNICODE[38874] := 16#EECA;
   // GBK_TO_UNICODE[38875] := 16#948D;
   // GBK_TO_UNICODE[38876] := 16#EECB;
   // GBK_TO_UNICODE[38877] := 16#948F;
   // GBK_TO_UNICODE[38878] := 16#EECC;
   // GBK_TO_UNICODE[38879] := 16#9490;
   // GBK_TO_UNICODE[38880] := 16#EECD;
   // GBK_TO_UNICODE[38881] := 16#9494;
   // GBK_TO_UNICODE[38882] := 16#EECE;
   // GBK_TO_UNICODE[38883] := 16#9497;
   // GBK_TO_UNICODE[38884] := 16#EECF;
   // GBK_TO_UNICODE[38885] := 16#9495;
   // GBK_TO_UNICODE[38886] := 16#EED0;
   // GBK_TO_UNICODE[38887] := 16#949A;
   // GBK_TO_UNICODE[38888] := 16#EED1;
   // GBK_TO_UNICODE[38889] := 16#949B;
   // GBK_TO_UNICODE[38890] := 16#EED2;
   // GBK_TO_UNICODE[38891] := 16#949C;
   // GBK_TO_UNICODE[38892] := 16#EED3;
   // GBK_TO_UNICODE[38893] := 16#94A3;
   // GBK_TO_UNICODE[38894] := 16#EED4;
   // GBK_TO_UNICODE[38895] := 16#94A4;
   // GBK_TO_UNICODE[38896] := 16#EED5;
   // GBK_TO_UNICODE[38897] := 16#94AB;
   // GBK_TO_UNICODE[38898] := 16#EED6;
   // GBK_TO_UNICODE[38899] := 16#94AA;
   // GBK_TO_UNICODE[38900] := 16#EED7;
   // GBK_TO_UNICODE[38901] := 16#94AD;
   // GBK_TO_UNICODE[38902] := 16#EED8;
   // GBK_TO_UNICODE[38903] := 16#94AC;
   // GBK_TO_UNICODE[38904] := 16#EED9;
   // GBK_TO_UNICODE[38905] := 16#94AF;
   // GBK_TO_UNICODE[38906] := 16#EEDA;
   // GBK_TO_UNICODE[38907] := 16#94B0;
   // GBK_TO_UNICODE[38908] := 16#EEDB;
   // GBK_TO_UNICODE[38909] := 16#94B2;
   // GBK_TO_UNICODE[38910] := 16#EEDC;
   // GBK_TO_UNICODE[38911] := 16#94B4;
   // GBK_TO_UNICODE[38912] := 16#EEDD;
   // GBK_TO_UNICODE[38913] := 16#94B6;
   // GBK_TO_UNICODE[38914] := 16#EEDE;
   // GBK_TO_UNICODE[38915] := 16#94B7;
   // GBK_TO_UNICODE[38916] := 16#EEDF;
   // GBK_TO_UNICODE[38917] := 16#94B8;
   // GBK_TO_UNICODE[38918] := 16#EEE0;
   // GBK_TO_UNICODE[38919] := 16#94B9;
   // GBK_TO_UNICODE[38920] := 16#EEE1;
   // GBK_TO_UNICODE[38921] := 16#94BA;
   // GBK_TO_UNICODE[38922] := 16#EEE2;
   // GBK_TO_UNICODE[38923] := 16#94BC;
   // GBK_TO_UNICODE[38924] := 16#EEE3;
   // GBK_TO_UNICODE[38925] := 16#94BD;
   // GBK_TO_UNICODE[38926] := 16#EEE4;
   // GBK_TO_UNICODE[38927] := 16#94BF;
   // GBK_TO_UNICODE[38928] := 16#EEE5;
   // GBK_TO_UNICODE[38929] := 16#94C4;
   // GBK_TO_UNICODE[38930] := 16#EEE6;
   // GBK_TO_UNICODE[38931] := 16#94C8;
   // GBK_TO_UNICODE[38932] := 16#EEE7;
   // GBK_TO_UNICODE[38933] := 16#94C9;
   // GBK_TO_UNICODE[38934] := 16#EEE8;
   // GBK_TO_UNICODE[38935] := 16#94CA;
   // GBK_TO_UNICODE[38936] := 16#EEE9;
   // GBK_TO_UNICODE[38937] := 16#94CB;
   // GBK_TO_UNICODE[38938] := 16#EEEA;
   // GBK_TO_UNICODE[38939] := 16#94CC;
   // GBK_TO_UNICODE[38940] := 16#EEEB;
   // GBK_TO_UNICODE[38941] := 16#94CD;
   // GBK_TO_UNICODE[38942] := 16#EEEC;
   // GBK_TO_UNICODE[38943] := 16#94CE;
   // GBK_TO_UNICODE[38944] := 16#EEED;
   // GBK_TO_UNICODE[38945] := 16#94D0;
   // GBK_TO_UNICODE[38946] := 16#EEEE;
   // GBK_TO_UNICODE[38947] := 16#94D1;
   // GBK_TO_UNICODE[38948] := 16#EEEF;
   // GBK_TO_UNICODE[38949] := 16#94D2;
   // GBK_TO_UNICODE[38950] := 16#EEF0;
   // GBK_TO_UNICODE[38951] := 16#94D5;
   // GBK_TO_UNICODE[38952] := 16#EEF1;
   // GBK_TO_UNICODE[38953] := 16#94D6;
   // GBK_TO_UNICODE[38954] := 16#EEF2;
   // GBK_TO_UNICODE[38955] := 16#94D7;
   // GBK_TO_UNICODE[38956] := 16#EEF3;
   // GBK_TO_UNICODE[38957] := 16#94D9;
   // GBK_TO_UNICODE[38958] := 16#EEF4;
   // GBK_TO_UNICODE[38959] := 16#94D8;
   // GBK_TO_UNICODE[38960] := 16#EEF5;
   // GBK_TO_UNICODE[38961] := 16#94DB;
   // GBK_TO_UNICODE[38962] := 16#EEF6;
   // GBK_TO_UNICODE[38963] := 16#94DE;
   // GBK_TO_UNICODE[38964] := 16#EEF7;
   // GBK_TO_UNICODE[38965] := 16#94DF;
   // GBK_TO_UNICODE[38966] := 16#EEF8;
   // GBK_TO_UNICODE[38967] := 16#94E0;
   // GBK_TO_UNICODE[38968] := 16#EEF9;
   // GBK_TO_UNICODE[38969] := 16#94E2;
   // GBK_TO_UNICODE[38970] := 16#EEFA;
   // GBK_TO_UNICODE[38971] := 16#94E4;
   // GBK_TO_UNICODE[38972] := 16#EEFB;
   // GBK_TO_UNICODE[38973] := 16#94E5;
   // GBK_TO_UNICODE[38974] := 16#EEFC;
   // GBK_TO_UNICODE[38975] := 16#94E7;
   // GBK_TO_UNICODE[38976] := 16#EEFD;
   // GBK_TO_UNICODE[38977] := 16#94E8;
   // GBK_TO_UNICODE[38978] := 16#EEFE;
   // GBK_TO_UNICODE[38979] := 16#94EA;
   // GBK_TO_UNICODE[38980] := 16#EF40;
   // GBK_TO_UNICODE[38981] := 16#986F;
   // GBK_TO_UNICODE[38982] := 16#EF41;
   // GBK_TO_UNICODE[38983] := 16#9870;
   // GBK_TO_UNICODE[38984] := 16#EF42;
   // GBK_TO_UNICODE[38985] := 16#9871;
   // GBK_TO_UNICODE[38986] := 16#EF43;
   // GBK_TO_UNICODE[38987] := 16#9872;
   // GBK_TO_UNICODE[38988] := 16#EF44;
   // GBK_TO_UNICODE[38989] := 16#9873;
   // GBK_TO_UNICODE[38990] := 16#EF45;
   // GBK_TO_UNICODE[38991] := 16#9874;
   // GBK_TO_UNICODE[38992] := 16#EF46;
   // GBK_TO_UNICODE[38993] := 16#988B;
   // GBK_TO_UNICODE[38994] := 16#EF47;
   // GBK_TO_UNICODE[38995] := 16#988E;
   // GBK_TO_UNICODE[38996] := 16#EF48;
   // GBK_TO_UNICODE[38997] := 16#9892;
   // GBK_TO_UNICODE[38998] := 16#EF49;
   // GBK_TO_UNICODE[38999] := 16#9895;
   // GBK_TO_UNICODE[39000] := 16#EF4A;
   // GBK_TO_UNICODE[39001] := 16#9899;
   // GBK_TO_UNICODE[39002] := 16#EF4B;
   // GBK_TO_UNICODE[39003] := 16#98A3;
   // GBK_TO_UNICODE[39004] := 16#EF4C;
   // GBK_TO_UNICODE[39005] := 16#98A8;
   // GBK_TO_UNICODE[39006] := 16#EF4D;
   // GBK_TO_UNICODE[39007] := 16#98A9;
   // GBK_TO_UNICODE[39008] := 16#EF4E;
   // GBK_TO_UNICODE[39009] := 16#98AA;
   // GBK_TO_UNICODE[39010] := 16#EF4F;
   // GBK_TO_UNICODE[39011] := 16#98AB;
   // GBK_TO_UNICODE[39012] := 16#EF50;
   // GBK_TO_UNICODE[39013] := 16#98AC;
   // GBK_TO_UNICODE[39014] := 16#EF51;
   // GBK_TO_UNICODE[39015] := 16#98AD;
   // GBK_TO_UNICODE[39016] := 16#EF52;
   // GBK_TO_UNICODE[39017] := 16#98AE;
   // GBK_TO_UNICODE[39018] := 16#EF53;
   // GBK_TO_UNICODE[39019] := 16#98AF;
   // GBK_TO_UNICODE[39020] := 16#EF54;
   // GBK_TO_UNICODE[39021] := 16#98B0;
   // GBK_TO_UNICODE[39022] := 16#EF55;
   // GBK_TO_UNICODE[39023] := 16#98B1;
   // GBK_TO_UNICODE[39024] := 16#EF56;
   // GBK_TO_UNICODE[39025] := 16#98B2;
   // GBK_TO_UNICODE[39026] := 16#EF57;
   // GBK_TO_UNICODE[39027] := 16#98B3;
   // GBK_TO_UNICODE[39028] := 16#EF58;
   // GBK_TO_UNICODE[39029] := 16#98B4;
   // GBK_TO_UNICODE[39030] := 16#EF59;
   // GBK_TO_UNICODE[39031] := 16#98B5;
   // GBK_TO_UNICODE[39032] := 16#EF5A;
   // GBK_TO_UNICODE[39033] := 16#98B6;
   // GBK_TO_UNICODE[39034] := 16#EF5B;
   // GBK_TO_UNICODE[39035] := 16#98B7;
   // GBK_TO_UNICODE[39036] := 16#EF5C;
   // GBK_TO_UNICODE[39037] := 16#98B8;
   // GBK_TO_UNICODE[39038] := 16#EF5D;
   // GBK_TO_UNICODE[39039] := 16#98B9;
   // GBK_TO_UNICODE[39040] := 16#EF5E;
   // GBK_TO_UNICODE[39041] := 16#98BA;
   // GBK_TO_UNICODE[39042] := 16#EF5F;
   // GBK_TO_UNICODE[39043] := 16#98BB;
   // GBK_TO_UNICODE[39044] := 16#EF60;
   // GBK_TO_UNICODE[39045] := 16#98BC;
   // GBK_TO_UNICODE[39046] := 16#EF61;
   // GBK_TO_UNICODE[39047] := 16#98BD;
   // GBK_TO_UNICODE[39048] := 16#EF62;
   // GBK_TO_UNICODE[39049] := 16#98BE;
   // GBK_TO_UNICODE[39050] := 16#EF63;
   // GBK_TO_UNICODE[39051] := 16#98BF;
   // GBK_TO_UNICODE[39052] := 16#EF64;
   // GBK_TO_UNICODE[39053] := 16#98C0;
   // GBK_TO_UNICODE[39054] := 16#EF65;
   // GBK_TO_UNICODE[39055] := 16#98C1;
   // GBK_TO_UNICODE[39056] := 16#EF66;
   // GBK_TO_UNICODE[39057] := 16#98C2;
   // GBK_TO_UNICODE[39058] := 16#EF67;
   // GBK_TO_UNICODE[39059] := 16#98C3;
   // GBK_TO_UNICODE[39060] := 16#EF68;
   // GBK_TO_UNICODE[39061] := 16#98C4;
   // GBK_TO_UNICODE[39062] := 16#EF69;
   // GBK_TO_UNICODE[39063] := 16#98C5;
   // GBK_TO_UNICODE[39064] := 16#EF6A;
   // GBK_TO_UNICODE[39065] := 16#98C6;
   // GBK_TO_UNICODE[39066] := 16#EF6B;
   // GBK_TO_UNICODE[39067] := 16#98C7;
   // GBK_TO_UNICODE[39068] := 16#EF6C;
   // GBK_TO_UNICODE[39069] := 16#98C8;
   // GBK_TO_UNICODE[39070] := 16#EF6D;
   // GBK_TO_UNICODE[39071] := 16#98C9;
   // GBK_TO_UNICODE[39072] := 16#EF6E;
   // GBK_TO_UNICODE[39073] := 16#98CA;
   // GBK_TO_UNICODE[39074] := 16#EF6F;
   // GBK_TO_UNICODE[39075] := 16#98CB;
   // GBK_TO_UNICODE[39076] := 16#EF70;
   // GBK_TO_UNICODE[39077] := 16#98CC;
   // GBK_TO_UNICODE[39078] := 16#EF71;
   // GBK_TO_UNICODE[39079] := 16#98CD;
   // GBK_TO_UNICODE[39080] := 16#EF72;
   // GBK_TO_UNICODE[39081] := 16#98CF;
   // GBK_TO_UNICODE[39082] := 16#EF73;
   // GBK_TO_UNICODE[39083] := 16#98D0;
   // GBK_TO_UNICODE[39084] := 16#EF74;
   // GBK_TO_UNICODE[39085] := 16#98D4;
   // GBK_TO_UNICODE[39086] := 16#EF75;
   // GBK_TO_UNICODE[39087] := 16#98D6;
   // GBK_TO_UNICODE[39088] := 16#EF76;
   // GBK_TO_UNICODE[39089] := 16#98D7;
   // GBK_TO_UNICODE[39090] := 16#EF77;
   // GBK_TO_UNICODE[39091] := 16#98DB;
   // GBK_TO_UNICODE[39092] := 16#EF78;
   // GBK_TO_UNICODE[39093] := 16#98DC;
   // GBK_TO_UNICODE[39094] := 16#EF79;
   // GBK_TO_UNICODE[39095] := 16#98DD;
   // GBK_TO_UNICODE[39096] := 16#EF7A;
   // GBK_TO_UNICODE[39097] := 16#98E0;
   // GBK_TO_UNICODE[39098] := 16#EF7B;
   // GBK_TO_UNICODE[39099] := 16#98E1;
   // GBK_TO_UNICODE[39100] := 16#EF7C;
   // GBK_TO_UNICODE[39101] := 16#98E2;
   // GBK_TO_UNICODE[39102] := 16#EF7D;
   // GBK_TO_UNICODE[39103] := 16#98E3;
   // GBK_TO_UNICODE[39104] := 16#EF7E;
   // GBK_TO_UNICODE[39105] := 16#98E4;
   // GBK_TO_UNICODE[39106] := 16#EF80;
   // GBK_TO_UNICODE[39107] := 16#98E5;
   // GBK_TO_UNICODE[39108] := 16#EF81;
   // GBK_TO_UNICODE[39109] := 16#98E6;
   // GBK_TO_UNICODE[39110] := 16#EF82;
   // GBK_TO_UNICODE[39111] := 16#98E9;
   // GBK_TO_UNICODE[39112] := 16#EF83;
   // GBK_TO_UNICODE[39113] := 16#98EA;
   // GBK_TO_UNICODE[39114] := 16#EF84;
   // GBK_TO_UNICODE[39115] := 16#98EB;
   // GBK_TO_UNICODE[39116] := 16#EF85;
   // GBK_TO_UNICODE[39117] := 16#98EC;
   // GBK_TO_UNICODE[39118] := 16#EF86;
   // GBK_TO_UNICODE[39119] := 16#98ED;
   // GBK_TO_UNICODE[39120] := 16#EF87;
   // GBK_TO_UNICODE[39121] := 16#98EE;
   // GBK_TO_UNICODE[39122] := 16#EF88;
   // GBK_TO_UNICODE[39123] := 16#98EF;
   // GBK_TO_UNICODE[39124] := 16#EF89;
   // GBK_TO_UNICODE[39125] := 16#98F0;
   // GBK_TO_UNICODE[39126] := 16#EF8A;
   // GBK_TO_UNICODE[39127] := 16#98F1;
   // GBK_TO_UNICODE[39128] := 16#EF8B;
   // GBK_TO_UNICODE[39129] := 16#98F2;
   // GBK_TO_UNICODE[39130] := 16#EF8C;
   // GBK_TO_UNICODE[39131] := 16#98F3;
   // GBK_TO_UNICODE[39132] := 16#EF8D;
   // GBK_TO_UNICODE[39133] := 16#98F4;
   // GBK_TO_UNICODE[39134] := 16#EF8E;
   // GBK_TO_UNICODE[39135] := 16#98F5;
   // GBK_TO_UNICODE[39136] := 16#EF8F;
   // GBK_TO_UNICODE[39137] := 16#98F6;
   // GBK_TO_UNICODE[39138] := 16#EF90;
   // GBK_TO_UNICODE[39139] := 16#98F7;
   // GBK_TO_UNICODE[39140] := 16#EF91;
   // GBK_TO_UNICODE[39141] := 16#98F8;
   // GBK_TO_UNICODE[39142] := 16#EF92;
   // GBK_TO_UNICODE[39143] := 16#98F9;
   // GBK_TO_UNICODE[39144] := 16#EF93;
   // GBK_TO_UNICODE[39145] := 16#98FA;
   // GBK_TO_UNICODE[39146] := 16#EF94;
   // GBK_TO_UNICODE[39147] := 16#98FB;
   // GBK_TO_UNICODE[39148] := 16#EF95;
   // GBK_TO_UNICODE[39149] := 16#98FC;
   // GBK_TO_UNICODE[39150] := 16#EF96;
   // GBK_TO_UNICODE[39151] := 16#98FD;
   // GBK_TO_UNICODE[39152] := 16#EF97;
   // GBK_TO_UNICODE[39153] := 16#98FE;
   // GBK_TO_UNICODE[39154] := 16#EF98;
   // GBK_TO_UNICODE[39155] := 16#98FF;
   // GBK_TO_UNICODE[39156] := 16#EF99;
   // GBK_TO_UNICODE[39157] := 16#9900;
   // GBK_TO_UNICODE[39158] := 16#EF9A;
   // GBK_TO_UNICODE[39159] := 16#9901;
   // GBK_TO_UNICODE[39160] := 16#EF9B;
   // GBK_TO_UNICODE[39161] := 16#9902;
   // GBK_TO_UNICODE[39162] := 16#EF9C;
   // GBK_TO_UNICODE[39163] := 16#9903;
   // GBK_TO_UNICODE[39164] := 16#EF9D;
   // GBK_TO_UNICODE[39165] := 16#9904;
   // GBK_TO_UNICODE[39166] := 16#EF9E;
   // GBK_TO_UNICODE[39167] := 16#9905;
   // GBK_TO_UNICODE[39168] := 16#EF9F;
   // GBK_TO_UNICODE[39169] := 16#9906;
   // GBK_TO_UNICODE[39170] := 16#EFA0;
   // GBK_TO_UNICODE[39171] := 16#9907;
   // GBK_TO_UNICODE[39172] := 16#EFA1;
   // GBK_TO_UNICODE[39173] := 16#94E9;
   // GBK_TO_UNICODE[39174] := 16#EFA2;
   // GBK_TO_UNICODE[39175] := 16#94EB;
   // GBK_TO_UNICODE[39176] := 16#EFA3;
   // GBK_TO_UNICODE[39177] := 16#94EE;
   // GBK_TO_UNICODE[39178] := 16#EFA4;
   // GBK_TO_UNICODE[39179] := 16#94EF;
   // GBK_TO_UNICODE[39180] := 16#EFA5;
   // GBK_TO_UNICODE[39181] := 16#94F3;
   // GBK_TO_UNICODE[39182] := 16#EFA6;
   // GBK_TO_UNICODE[39183] := 16#94F4;
   // GBK_TO_UNICODE[39184] := 16#EFA7;
   // GBK_TO_UNICODE[39185] := 16#94F5;
   // GBK_TO_UNICODE[39186] := 16#EFA8;
   // GBK_TO_UNICODE[39187] := 16#94F7;
   // GBK_TO_UNICODE[39188] := 16#EFA9;
   // GBK_TO_UNICODE[39189] := 16#94F9;
   // GBK_TO_UNICODE[39190] := 16#EFAA;
   // GBK_TO_UNICODE[39191] := 16#94FC;
   // GBK_TO_UNICODE[39192] := 16#EFAB;
   // GBK_TO_UNICODE[39193] := 16#94FD;
   // GBK_TO_UNICODE[39194] := 16#EFAC;
   // GBK_TO_UNICODE[39195] := 16#94FF;
   // GBK_TO_UNICODE[39196] := 16#EFAD;
   // GBK_TO_UNICODE[39197] := 16#9503;
   // GBK_TO_UNICODE[39198] := 16#EFAE;
   // GBK_TO_UNICODE[39199] := 16#9502;
   // GBK_TO_UNICODE[39200] := 16#EFAF;
   // GBK_TO_UNICODE[39201] := 16#9506;
   // GBK_TO_UNICODE[39202] := 16#EFB0;
   // GBK_TO_UNICODE[39203] := 16#9507;
   // GBK_TO_UNICODE[39204] := 16#EFB1;
   // GBK_TO_UNICODE[39205] := 16#9509;
   // GBK_TO_UNICODE[39206] := 16#EFB2;
   // GBK_TO_UNICODE[39207] := 16#950A;
   // GBK_TO_UNICODE[39208] := 16#EFB3;
   // GBK_TO_UNICODE[39209] := 16#950D;
   // GBK_TO_UNICODE[39210] := 16#EFB4;
   // GBK_TO_UNICODE[39211] := 16#950E;
   // GBK_TO_UNICODE[39212] := 16#EFB5;
   // GBK_TO_UNICODE[39213] := 16#950F;
   // GBK_TO_UNICODE[39214] := 16#EFB6;
   // GBK_TO_UNICODE[39215] := 16#9512;
   // GBK_TO_UNICODE[39216] := 16#EFB7;
   // GBK_TO_UNICODE[39217] := 16#9513;
   // GBK_TO_UNICODE[39218] := 16#EFB8;
   // GBK_TO_UNICODE[39219] := 16#9514;
   // GBK_TO_UNICODE[39220] := 16#EFB9;
   // GBK_TO_UNICODE[39221] := 16#9515;
   // GBK_TO_UNICODE[39222] := 16#EFBA;
   // GBK_TO_UNICODE[39223] := 16#9516;
   // GBK_TO_UNICODE[39224] := 16#EFBB;
   // GBK_TO_UNICODE[39225] := 16#9518;
   // GBK_TO_UNICODE[39226] := 16#EFBC;
   // GBK_TO_UNICODE[39227] := 16#951B;
   // GBK_TO_UNICODE[39228] := 16#EFBD;
   // GBK_TO_UNICODE[39229] := 16#951D;
   // GBK_TO_UNICODE[39230] := 16#EFBE;
   // GBK_TO_UNICODE[39231] := 16#951E;
   // GBK_TO_UNICODE[39232] := 16#EFBF;
   // GBK_TO_UNICODE[39233] := 16#951F;
   // GBK_TO_UNICODE[39234] := 16#EFC0;
   // GBK_TO_UNICODE[39235] := 16#9522;
   // GBK_TO_UNICODE[39236] := 16#EFC1;
   // GBK_TO_UNICODE[39237] := 16#952A;
   // GBK_TO_UNICODE[39238] := 16#EFC2;
   // GBK_TO_UNICODE[39239] := 16#952B;
   // GBK_TO_UNICODE[39240] := 16#EFC3;
   // GBK_TO_UNICODE[39241] := 16#9529;
   // GBK_TO_UNICODE[39242] := 16#EFC4;
   // GBK_TO_UNICODE[39243] := 16#952C;
   // GBK_TO_UNICODE[39244] := 16#EFC5;
   // GBK_TO_UNICODE[39245] := 16#9531;
   // GBK_TO_UNICODE[39246] := 16#EFC6;
   // GBK_TO_UNICODE[39247] := 16#9532;
   // GBK_TO_UNICODE[39248] := 16#EFC7;
   // GBK_TO_UNICODE[39249] := 16#9534;
   // GBK_TO_UNICODE[39250] := 16#EFC8;
   // GBK_TO_UNICODE[39251] := 16#9536;
   // GBK_TO_UNICODE[39252] := 16#EFC9;
   // GBK_TO_UNICODE[39253] := 16#9537;
   // GBK_TO_UNICODE[39254] := 16#EFCA;
   // GBK_TO_UNICODE[39255] := 16#9538;
   // GBK_TO_UNICODE[39256] := 16#EFCB;
   // GBK_TO_UNICODE[39257] := 16#953C;
   // GBK_TO_UNICODE[39258] := 16#EFCC;
   // GBK_TO_UNICODE[39259] := 16#953E;
   // GBK_TO_UNICODE[39260] := 16#EFCD;
   // GBK_TO_UNICODE[39261] := 16#953F;
   // GBK_TO_UNICODE[39262] := 16#EFCE;
   // GBK_TO_UNICODE[39263] := 16#9542;
   // GBK_TO_UNICODE[39264] := 16#EFCF;
   // GBK_TO_UNICODE[39265] := 16#9535;
   // GBK_TO_UNICODE[39266] := 16#EFD0;
   // GBK_TO_UNICODE[39267] := 16#9544;
   // GBK_TO_UNICODE[39268] := 16#EFD1;
   // GBK_TO_UNICODE[39269] := 16#9545;
   // GBK_TO_UNICODE[39270] := 16#EFD2;
   // GBK_TO_UNICODE[39271] := 16#9546;
   // GBK_TO_UNICODE[39272] := 16#EFD3;
   // GBK_TO_UNICODE[39273] := 16#9549;
   // GBK_TO_UNICODE[39274] := 16#EFD4;
   // GBK_TO_UNICODE[39275] := 16#954C;
   // GBK_TO_UNICODE[39276] := 16#EFD5;
   // GBK_TO_UNICODE[39277] := 16#954E;
   // GBK_TO_UNICODE[39278] := 16#EFD6;
   // GBK_TO_UNICODE[39279] := 16#954F;
   // GBK_TO_UNICODE[39280] := 16#EFD7;
   // GBK_TO_UNICODE[39281] := 16#9552;
   // GBK_TO_UNICODE[39282] := 16#EFD8;
   // GBK_TO_UNICODE[39283] := 16#9553;
   // GBK_TO_UNICODE[39284] := 16#EFD9;
   // GBK_TO_UNICODE[39285] := 16#9554;
   // GBK_TO_UNICODE[39286] := 16#EFDA;
   // GBK_TO_UNICODE[39287] := 16#9556;
   // GBK_TO_UNICODE[39288] := 16#EFDB;
   // GBK_TO_UNICODE[39289] := 16#9557;
   // GBK_TO_UNICODE[39290] := 16#EFDC;
   // GBK_TO_UNICODE[39291] := 16#9558;
   // GBK_TO_UNICODE[39292] := 16#EFDD;
   // GBK_TO_UNICODE[39293] := 16#9559;
   // GBK_TO_UNICODE[39294] := 16#EFDE;
   // GBK_TO_UNICODE[39295] := 16#955B;
   // GBK_TO_UNICODE[39296] := 16#EFDF;
   // GBK_TO_UNICODE[39297] := 16#955E;
   // GBK_TO_UNICODE[39298] := 16#EFE0;
   // GBK_TO_UNICODE[39299] := 16#955F;
   // GBK_TO_UNICODE[39300] := 16#EFE1;
   // GBK_TO_UNICODE[39301] := 16#955D;
   // GBK_TO_UNICODE[39302] := 16#EFE2;
   // GBK_TO_UNICODE[39303] := 16#9561;
   // GBK_TO_UNICODE[39304] := 16#EFE3;
   // GBK_TO_UNICODE[39305] := 16#9562;
   // GBK_TO_UNICODE[39306] := 16#EFE4;
   // GBK_TO_UNICODE[39307] := 16#9564;
   // GBK_TO_UNICODE[39308] := 16#EFE5;
   // GBK_TO_UNICODE[39309] := 16#9565;
   // GBK_TO_UNICODE[39310] := 16#EFE6;
   // GBK_TO_UNICODE[39311] := 16#9566;
   // GBK_TO_UNICODE[39312] := 16#EFE7;
   // GBK_TO_UNICODE[39313] := 16#9567;
   // GBK_TO_UNICODE[39314] := 16#EFE8;
   // GBK_TO_UNICODE[39315] := 16#9568;
   // GBK_TO_UNICODE[39316] := 16#EFE9;
   // GBK_TO_UNICODE[39317] := 16#9569;
   // GBK_TO_UNICODE[39318] := 16#EFEA;
   // GBK_TO_UNICODE[39319] := 16#956A;
   // GBK_TO_UNICODE[39320] := 16#EFEB;
   // GBK_TO_UNICODE[39321] := 16#956B;
   // GBK_TO_UNICODE[39322] := 16#EFEC;
   // GBK_TO_UNICODE[39323] := 16#956C;
   // GBK_TO_UNICODE[39324] := 16#EFED;
   // GBK_TO_UNICODE[39325] := 16#956F;
   // GBK_TO_UNICODE[39326] := 16#EFEE;
   // GBK_TO_UNICODE[39327] := 16#9571;
   // GBK_TO_UNICODE[39328] := 16#EFEF;
   // GBK_TO_UNICODE[39329] := 16#9572;
   // GBK_TO_UNICODE[39330] := 16#EFF0;
   // GBK_TO_UNICODE[39331] := 16#9573;
   // GBK_TO_UNICODE[39332] := 16#EFF1;
   // GBK_TO_UNICODE[39333] := 16#953A;
   // GBK_TO_UNICODE[39334] := 16#EFF2;
   // GBK_TO_UNICODE[39335] := 16#77E7;
   // GBK_TO_UNICODE[39336] := 16#EFF3;
   // GBK_TO_UNICODE[39337] := 16#77EC;
   // GBK_TO_UNICODE[39338] := 16#EFF4;
   // GBK_TO_UNICODE[39339] := 16#96C9;
   // GBK_TO_UNICODE[39340] := 16#EFF5;
   // GBK_TO_UNICODE[39341] := 16#79D5;
   // GBK_TO_UNICODE[39342] := 16#EFF6;
   // GBK_TO_UNICODE[39343] := 16#79ED;
   // GBK_TO_UNICODE[39344] := 16#EFF7;
   // GBK_TO_UNICODE[39345] := 16#79E3;
   // GBK_TO_UNICODE[39346] := 16#EFF8;
   // GBK_TO_UNICODE[39347] := 16#79EB;
   // GBK_TO_UNICODE[39348] := 16#EFF9;
   // GBK_TO_UNICODE[39349] := 16#7A06;
   // GBK_TO_UNICODE[39350] := 16#EFFA;
   // GBK_TO_UNICODE[39351] := 16#5D47;
   // GBK_TO_UNICODE[39352] := 16#EFFB;
   // GBK_TO_UNICODE[39353] := 16#7A03;
   // GBK_TO_UNICODE[39354] := 16#EFFC;
   // GBK_TO_UNICODE[39355] := 16#7A02;
   // GBK_TO_UNICODE[39356] := 16#EFFD;
   // GBK_TO_UNICODE[39357] := 16#7A1E;
   // GBK_TO_UNICODE[39358] := 16#EFFE;
   // GBK_TO_UNICODE[39359] := 16#7A14;
   // GBK_TO_UNICODE[39360] := 16#F040;
   // GBK_TO_UNICODE[39361] := 16#9908;
   // GBK_TO_UNICODE[39362] := 16#F041;
   // GBK_TO_UNICODE[39363] := 16#9909;
   // GBK_TO_UNICODE[39364] := 16#F042;
   // GBK_TO_UNICODE[39365] := 16#990A;
   // GBK_TO_UNICODE[39366] := 16#F043;
   // GBK_TO_UNICODE[39367] := 16#990B;
   // GBK_TO_UNICODE[39368] := 16#F044;
   // GBK_TO_UNICODE[39369] := 16#990C;
   // GBK_TO_UNICODE[39370] := 16#F045;
   // GBK_TO_UNICODE[39371] := 16#990E;
   // GBK_TO_UNICODE[39372] := 16#F046;
   // GBK_TO_UNICODE[39373] := 16#990F;
   // GBK_TO_UNICODE[39374] := 16#F047;
   // GBK_TO_UNICODE[39375] := 16#9911;
   // GBK_TO_UNICODE[39376] := 16#F048;
   // GBK_TO_UNICODE[39377] := 16#9912;
   // GBK_TO_UNICODE[39378] := 16#F049;
   // GBK_TO_UNICODE[39379] := 16#9913;
   // GBK_TO_UNICODE[39380] := 16#F04A;
   // GBK_TO_UNICODE[39381] := 16#9914;
   // GBK_TO_UNICODE[39382] := 16#F04B;
   // GBK_TO_UNICODE[39383] := 16#9915;
   // GBK_TO_UNICODE[39384] := 16#F04C;
   // GBK_TO_UNICODE[39385] := 16#9916;
   // GBK_TO_UNICODE[39386] := 16#F04D;
   // GBK_TO_UNICODE[39387] := 16#9917;
   // GBK_TO_UNICODE[39388] := 16#F04E;
   // GBK_TO_UNICODE[39389] := 16#9918;
   // GBK_TO_UNICODE[39390] := 16#F04F;
   // GBK_TO_UNICODE[39391] := 16#9919;
   // GBK_TO_UNICODE[39392] := 16#F050;
   // GBK_TO_UNICODE[39393] := 16#991A;
   // GBK_TO_UNICODE[39394] := 16#F051;
   // GBK_TO_UNICODE[39395] := 16#991B;
   // GBK_TO_UNICODE[39396] := 16#F052;
   // GBK_TO_UNICODE[39397] := 16#991C;
   // GBK_TO_UNICODE[39398] := 16#F053;
   // GBK_TO_UNICODE[39399] := 16#991D;
   // GBK_TO_UNICODE[39400] := 16#F054;
   // GBK_TO_UNICODE[39401] := 16#991E;
   // GBK_TO_UNICODE[39402] := 16#F055;
   // GBK_TO_UNICODE[39403] := 16#991F;
   // GBK_TO_UNICODE[39404] := 16#F056;
   // GBK_TO_UNICODE[39405] := 16#9920;
   // GBK_TO_UNICODE[39406] := 16#F057;
   // GBK_TO_UNICODE[39407] := 16#9921;
   // GBK_TO_UNICODE[39408] := 16#F058;
   // GBK_TO_UNICODE[39409] := 16#9922;
   // GBK_TO_UNICODE[39410] := 16#F059;
   // GBK_TO_UNICODE[39411] := 16#9923;
   // GBK_TO_UNICODE[39412] := 16#F05A;
   // GBK_TO_UNICODE[39413] := 16#9924;
   // GBK_TO_UNICODE[39414] := 16#F05B;
   // GBK_TO_UNICODE[39415] := 16#9925;
   // GBK_TO_UNICODE[39416] := 16#F05C;
   // GBK_TO_UNICODE[39417] := 16#9926;
   // GBK_TO_UNICODE[39418] := 16#F05D;
   // GBK_TO_UNICODE[39419] := 16#9927;
   // GBK_TO_UNICODE[39420] := 16#F05E;
   // GBK_TO_UNICODE[39421] := 16#9928;
   // GBK_TO_UNICODE[39422] := 16#F05F;
   // GBK_TO_UNICODE[39423] := 16#9929;
   // GBK_TO_UNICODE[39424] := 16#F060;
   // GBK_TO_UNICODE[39425] := 16#992A;
   // GBK_TO_UNICODE[39426] := 16#F061;
   // GBK_TO_UNICODE[39427] := 16#992B;
   // GBK_TO_UNICODE[39428] := 16#F062;
   // GBK_TO_UNICODE[39429] := 16#992C;
   // GBK_TO_UNICODE[39430] := 16#F063;
   // GBK_TO_UNICODE[39431] := 16#992D;
   // GBK_TO_UNICODE[39432] := 16#F064;
   // GBK_TO_UNICODE[39433] := 16#992F;
   // GBK_TO_UNICODE[39434] := 16#F065;
   // GBK_TO_UNICODE[39435] := 16#9930;
   // GBK_TO_UNICODE[39436] := 16#F066;
   // GBK_TO_UNICODE[39437] := 16#9931;
   // GBK_TO_UNICODE[39438] := 16#F067;
   // GBK_TO_UNICODE[39439] := 16#9932;
   // GBK_TO_UNICODE[39440] := 16#F068;
   // GBK_TO_UNICODE[39441] := 16#9933;
   // GBK_TO_UNICODE[39442] := 16#F069;
   // GBK_TO_UNICODE[39443] := 16#9934;
   // GBK_TO_UNICODE[39444] := 16#F06A;
   // GBK_TO_UNICODE[39445] := 16#9935;
   // GBK_TO_UNICODE[39446] := 16#F06B;
   // GBK_TO_UNICODE[39447] := 16#9936;
   // GBK_TO_UNICODE[39448] := 16#F06C;
   // GBK_TO_UNICODE[39449] := 16#9937;
   // GBK_TO_UNICODE[39450] := 16#F06D;
   // GBK_TO_UNICODE[39451] := 16#9938;
   // GBK_TO_UNICODE[39452] := 16#F06E;
   // GBK_TO_UNICODE[39453] := 16#9939;
   // GBK_TO_UNICODE[39454] := 16#F06F;
   // GBK_TO_UNICODE[39455] := 16#993A;
   // GBK_TO_UNICODE[39456] := 16#F070;
   // GBK_TO_UNICODE[39457] := 16#993B;
   // GBK_TO_UNICODE[39458] := 16#F071;
   // GBK_TO_UNICODE[39459] := 16#993C;
   // GBK_TO_UNICODE[39460] := 16#F072;
   // GBK_TO_UNICODE[39461] := 16#993D;
   // GBK_TO_UNICODE[39462] := 16#F073;
   // GBK_TO_UNICODE[39463] := 16#993E;
   // GBK_TO_UNICODE[39464] := 16#F074;
   // GBK_TO_UNICODE[39465] := 16#993F;
   // GBK_TO_UNICODE[39466] := 16#F075;
   // GBK_TO_UNICODE[39467] := 16#9940;
   // GBK_TO_UNICODE[39468] := 16#F076;
   // GBK_TO_UNICODE[39469] := 16#9941;
   // GBK_TO_UNICODE[39470] := 16#F077;
   // GBK_TO_UNICODE[39471] := 16#9942;
   // GBK_TO_UNICODE[39472] := 16#F078;
   // GBK_TO_UNICODE[39473] := 16#9943;
   // GBK_TO_UNICODE[39474] := 16#F079;
   // GBK_TO_UNICODE[39475] := 16#9944;
   // GBK_TO_UNICODE[39476] := 16#F07A;
   // GBK_TO_UNICODE[39477] := 16#9945;
   // GBK_TO_UNICODE[39478] := 16#F07B;
   // GBK_TO_UNICODE[39479] := 16#9946;
   // GBK_TO_UNICODE[39480] := 16#F07C;
   // GBK_TO_UNICODE[39481] := 16#9947;
   // GBK_TO_UNICODE[39482] := 16#F07D;
   // GBK_TO_UNICODE[39483] := 16#9948;
   // GBK_TO_UNICODE[39484] := 16#F07E;
   // GBK_TO_UNICODE[39485] := 16#9949;
   // GBK_TO_UNICODE[39486] := 16#F080;
   // GBK_TO_UNICODE[39487] := 16#994A;
   // GBK_TO_UNICODE[39488] := 16#F081;
   // GBK_TO_UNICODE[39489] := 16#994B;
   // GBK_TO_UNICODE[39490] := 16#F082;
   // GBK_TO_UNICODE[39491] := 16#994C;
   // GBK_TO_UNICODE[39492] := 16#F083;
   // GBK_TO_UNICODE[39493] := 16#994D;
   // GBK_TO_UNICODE[39494] := 16#F084;
   // GBK_TO_UNICODE[39495] := 16#994E;
   // GBK_TO_UNICODE[39496] := 16#F085;
   // GBK_TO_UNICODE[39497] := 16#994F;
   // GBK_TO_UNICODE[39498] := 16#F086;
   // GBK_TO_UNICODE[39499] := 16#9950;
   // GBK_TO_UNICODE[39500] := 16#F087;
   // GBK_TO_UNICODE[39501] := 16#9951;
   // GBK_TO_UNICODE[39502] := 16#F088;
   // GBK_TO_UNICODE[39503] := 16#9952;
   // GBK_TO_UNICODE[39504] := 16#F089;
   // GBK_TO_UNICODE[39505] := 16#9953;
   // GBK_TO_UNICODE[39506] := 16#F08A;
   // GBK_TO_UNICODE[39507] := 16#9956;
   // GBK_TO_UNICODE[39508] := 16#F08B;
   // GBK_TO_UNICODE[39509] := 16#9957;
   // GBK_TO_UNICODE[39510] := 16#F08C;
   // GBK_TO_UNICODE[39511] := 16#9958;
   // GBK_TO_UNICODE[39512] := 16#F08D;
   // GBK_TO_UNICODE[39513] := 16#9959;
   // GBK_TO_UNICODE[39514] := 16#F08E;
   // GBK_TO_UNICODE[39515] := 16#995A;
   // GBK_TO_UNICODE[39516] := 16#F08F;
   // GBK_TO_UNICODE[39517] := 16#995B;
   // GBK_TO_UNICODE[39518] := 16#F090;
   // GBK_TO_UNICODE[39519] := 16#995C;
   // GBK_TO_UNICODE[39520] := 16#F091;
   // GBK_TO_UNICODE[39521] := 16#995D;
   // GBK_TO_UNICODE[39522] := 16#F092;
   // GBK_TO_UNICODE[39523] := 16#995E;
   // GBK_TO_UNICODE[39524] := 16#F093;
   // GBK_TO_UNICODE[39525] := 16#995F;
   // GBK_TO_UNICODE[39526] := 16#F094;
   // GBK_TO_UNICODE[39527] := 16#9960;
   // GBK_TO_UNICODE[39528] := 16#F095;
   // GBK_TO_UNICODE[39529] := 16#9961;
   // GBK_TO_UNICODE[39530] := 16#F096;
   // GBK_TO_UNICODE[39531] := 16#9962;
   // GBK_TO_UNICODE[39532] := 16#F097;
   // GBK_TO_UNICODE[39533] := 16#9964;
   // GBK_TO_UNICODE[39534] := 16#F098;
   // GBK_TO_UNICODE[39535] := 16#9966;
   // GBK_TO_UNICODE[39536] := 16#F099;
   // GBK_TO_UNICODE[39537] := 16#9973;
   // GBK_TO_UNICODE[39538] := 16#F09A;
   // GBK_TO_UNICODE[39539] := 16#9978;
   // GBK_TO_UNICODE[39540] := 16#F09B;
   // GBK_TO_UNICODE[39541] := 16#9979;
   // GBK_TO_UNICODE[39542] := 16#F09C;
   // GBK_TO_UNICODE[39543] := 16#997B;
   // GBK_TO_UNICODE[39544] := 16#F09D;
   // GBK_TO_UNICODE[39545] := 16#997E;
   // GBK_TO_UNICODE[39546] := 16#F09E;
   // GBK_TO_UNICODE[39547] := 16#9982;
   // GBK_TO_UNICODE[39548] := 16#F09F;
   // GBK_TO_UNICODE[39549] := 16#9983;
   // GBK_TO_UNICODE[39550] := 16#F0A0;
   // GBK_TO_UNICODE[39551] := 16#9989;
   // GBK_TO_UNICODE[39552] := 16#F0A1;
   // GBK_TO_UNICODE[39553] := 16#7A39;
   // GBK_TO_UNICODE[39554] := 16#F0A2;
   // GBK_TO_UNICODE[39555] := 16#7A37;
   // GBK_TO_UNICODE[39556] := 16#F0A3;
   // GBK_TO_UNICODE[39557] := 16#7A51;
   // GBK_TO_UNICODE[39558] := 16#F0A4;
   // GBK_TO_UNICODE[39559] := 16#9ECF;
   // GBK_TO_UNICODE[39560] := 16#F0A5;
   // GBK_TO_UNICODE[39561] := 16#99A5;
   // GBK_TO_UNICODE[39562] := 16#F0A6;
   // GBK_TO_UNICODE[39563] := 16#7A70;
   // GBK_TO_UNICODE[39564] := 16#F0A7;
   // GBK_TO_UNICODE[39565] := 16#7688;
   // GBK_TO_UNICODE[39566] := 16#F0A8;
   // GBK_TO_UNICODE[39567] := 16#768E;
